	UF : 0, UT : 6,		CONFIG : 'N U T, 0, 0, 0',
	X =  94.552  mm,	Y =   -408.352  mm,	Z =   -258.182  mm,
	W =  90.000 deg,	P =   0.000 deg,	R =   90.000 deg
};
P[1225]{
   GP1:
	UF : 0, UT : 6,		CONFIG : 'N U T, 0, 0, 0',
	X =  95.294  mm,	Y =   -409.608  mm,	Z =   -258.283  mm,
	W =  90.000 deg,	P =   0.000 deg,	R =   90.000 deg
};
P[1226]{
   GP1:
	UF : 0, UT : 6,		CONFIG : 'N U T, 0, 0, 0',
	X =  95.758  mm,	Y =   -410.484  mm,	Z =   -258.027  mm,
	W =  90.000 deg,	P =   0.000 deg,	R =   90.000 deg
};
P[1227]{
   GP1:
	UF : 0, UT : 6,		CONFIG : 'N U T, 0, 0, 0',
	X =  97.788  mm,	Y =   -414.039  mm,	Z =   -257.885  mm,
	W =  90.000 deg,	P =   0.000 deg,	R =   90.000 deg
};
P[1228]{
   GP1:
	UF : 0, UT : 6,		CONFIG : 'N U T, 0, 0, 0',
	X =  98.420  mm,	Y =   -415.000  mm,	Z =   -258.363  mm,
	W =  90.000 deg,	P =   0.000 deg,	R =   90.000 deg
};
P[1229]{
   GP1:
	UF : 0, UT : 6,		CONFIG : 'N U T, 0, 0, 0',
	X =  98.908  mm,	Y =   -415.884  mm,	Z =   -258.225  mm,
	W =  90.000 deg,	P =   0.000 deg,	R =   90.000 deg
};
P[1230]{
   GP1:
	UF : 0, UT : 6,		CONFIG : 'N U T, 0, 0, 0',
	X =  99.222  mm,	Y =   -416.492  mm,	Z =   -257.998  mm,
	W =  90.000 deg,	P =   0.000 deg,	R =   90.000 deg
};
P[1231]{
   GP1:
	UF : 0, UT : 6,		CONFIG : 'N U T, 0, 0, 0',
	X =  99.637  mm,	Y =   -417.217  mm,	Z =   -257.979  mm,
	W =  90.000 deg,	P =   0.000 deg,	R =   90.000 deg
};
P[1232]{
   GP1:
	UF : 0, UT : 6,		CONFIG : 'N U T, 0, 0, 0',
	X =  100.678  mm,	Y =   -419.015  mm,	Z =   -257.989  mm,
	W =  90.000 deg,	P =   0.000 deg,	R =   90.000 deg
};
P[1233]{
   GP1:
	UF : 0, UT : 6,		CONFIG : 'N U T, 0, 0, 0',
	X =  102.165  mm,	Y =   -421.501  mm,	Z =   -258.308  mm,
	W =  90.000 deg,	P =   0.000 deg,	R =   90.000 deg
};
P[1234]{
   GP1:
	UF : 0, UT : 6,		CONFIG : 'N U T, 0, 0, 0',
	X =  102.557  mm,	Y =   -422.208  mm,	Z =   -258.207  mm,
	W =  90.000 deg,	P =   0.000 deg,	R =   90.000 deg
};
P[1235]{
   GP1:
	UF : 0, UT : 6,		CONFIG : 'N U T, 0, 0, 0',
	X =  103.682  mm,	Y =   -424.148  mm,	Z =   -258.237  mm,
	W =  90.000 deg,	P =   0.000 deg,	R =   90.000 deg
};
P[1236]{
   GP1:
	UF : 0, UT : 6,		CONFIG : 'N U T, 0, 0, 0',
	X =  104.838  mm,	Y =   -426.195  mm,	Z =   -258.076  mm,
	W =  90.000 deg,	P =   0.000 deg,	R =   90.000 deg
};
P[1237]{
   GP1:
	UF : 0, UT : 6,		CONFIG : 'N U T, 0, 0, 0',
	X =  106.776  mm,	Y =   -429.472  mm,	Z =   -258.366  mm,
	W =  90.000 deg,	P =   0.000 deg,	R =   90.000 deg
};
P[1238]{
   GP1:
	UF : 0, UT : 6,		CONFIG : 'N U T, 0, 0, 0',
	X =  107.228  mm,	Y =   -430.273  mm,	Z =   -258.299  mm,
	W =  90.000 deg,	P =   0.000 deg,	R =   90.000 deg
};
P[1239]{
   GP1:
	UF : 0, UT : 6,		CONFIG : 'N U T, 0, 0, 0',
	X =  108.043  mm,	Y =   -431.682  mm,	Z =   -258.309  mm,
	W =  90.000 deg,	P =   0.000 deg,	R =   90.000 deg
};
P[1240]{
   GP1:
	UF : 0, UT : 6,		CONFIG : 'N U T, 0, 0, 0',
	X =  108.614  mm,	Y =   -432.663  mm,	Z =   -258.336  mm,
	W =  90.000 deg,	P =   0.000 deg,	R =   90.000 deg
};
P[1241]{
   GP1:
	UF : 0, UT : 6,		CONFIG : 'N U T, 0, 0, 0',
	X =  110.290  mm,	Y =   -435.622  mm,	Z =   -258.135  mm,
	W =  90.000 deg,	P =   0.000 deg,	R =   90.000 deg
};
P[1242]{
   GP1:
	UF : 0, UT : 6,		CONFIG : 'N U T, 0, 0, 0',
	X =  110.941  mm,	Y =   -436.722  mm,	Z =   -258.230  mm,
	W =  90.000 deg,	P =   0.000 deg,	R =   90.000 deg
};
P[1243]{
   GP1:
	UF : 0, UT : 6,		CONFIG : 'N U T, 0, 0, 0',
	X =  112.232  mm,	Y =   -438.986  mm,	Z =   -258.130  mm,
	W =  90.000 deg,	P =   0.000 deg,	R =   90.000 deg
};
P[1244]{
   GP1:
	UF : 0, UT : 6,		CONFIG : 'N U T, 0, 0, 0',
	X =  113.189  mm,	Y =   -440.584  mm,	Z =   -258.341  mm,
	W =  90.000 deg,	P =   0.000 deg,	R =   90.000 deg
};
P[1245]{
   GP1:
	UF : 0, UT : 6,		CONFIG : 'N U T, 0, 0, 0',
	X =  114.856  mm,	Y =   -443.594  mm,	Z =   -257.910  mm,
	W =  90.000 deg,	P =   0.000 deg,	R =   90.000 deg
};
P[1246]{
   GP1:
	UF : 0, UT : 6,		CONFIG : 'N U T, 0, 0, 0',
	X =  115.439  mm,	Y =   -444.516  mm,	Z =   -258.220  mm,
	W =  90.000 deg,	P =   0.000 deg,	R =   90.000 deg
};
P[1247]{
   GP1:
	UF : 0, UT : 6,		CONFIG : 'N U T, 0, 0, 0',
	X =  115.884  mm,	Y =   -445.335  mm,	Z =   -258.046  mm,
	W =  90.000 deg,	P =   0.000 deg,	R =   90.000 deg
};
P[1248]{
   GP1:
	UF : 0, UT : 6,		CONFIG : 'N U T, 0, 0, 0',
	X =  116.583  mm,	Y =   -446.538  mm,	Z =   -258.073  mm,
	W =  90.000 deg,	P =   0.000 deg,	R =   90.000 deg
};
P[1249]{
   GP1:
	UF : 0, UT : 6,		CONFIG : 'N U T, 0, 0, 0',
	X =  117.265  mm,	Y =   -447.654  mm,	Z =   -258.308  mm,
	W =  90.000 deg,	P =   0.000 deg,	R =   90.000 deg
};
P[1250]{
   GP1:
	UF : 0, UT : 6,		CONFIG : 'N U T, 0, 0, 0',
	X =  118.172  mm,	Y =   -449.252  mm,	Z =   -258.213  mm,
	W =  90.000 deg,	P =   0.000 deg,	R =   90.000 deg
};
P[1251]{
   GP1:
	UF : 0, UT : 6,		CONFIG : 'N U T, 0, 0, 0',
	X =  119.589  mm,	Y =   -451.752  mm,	Z =   -258.047  mm,
	W =  90.000 deg,	P =   0.000 deg,	R =   90.000 deg
};
P[1252]{
   GP1:
	UF : 0, UT : 6,		CONFIG : 'N U T, 0, 0, 0',
	X =  120.416  mm,	Y =   -453.157  mm,	Z =   -258.146  mm,
	W =  90.000 deg,	P =   0.000 deg,	R =   90.000 deg
};
P[1253]{
   GP1:
	UF : 0, UT : 6,		CONFIG : 'N U T, 0, 0, 0',
	X =  120.901  mm,	Y =   -453.949  mm,	Z =   -258.320  mm,
	W =  90.000 deg,	P =   0.000 deg,	R =   90.000 deg
};
P[1254]{
   GP1:
	UF : 0, UT : 6,		CONFIG : 'N U T, 0, 0, 0',
	X =  121.824  mm,	Y =   -455.560  mm,	Z =   -258.271  mm,
	W =  90.000 deg,	P =   0.000 deg,	R =   90.000 deg
};
P[1255]{
   GP1:
	UF : 0, UT : 6,		CONFIG : 'N U T, 0, 0, 0',
	X =  122.704  mm,	Y =   -457.147  mm,	Z =   -258.049  mm,
	W =  90.000 deg,	P =   0.000 deg,	R =   90.000 deg
};
P[1256]{
   GP1:
	UF : 0, UT : 6,		CONFIG : 'N U T, 0, 0, 0',
	X =  123.451  mm,	Y =   -458.351  mm,	Z =   -258.366  mm,
	W =  90.000 deg,	P =   0.000 deg,	R =   90.000 deg
};
P[1257]{
   GP1:
	UF : 0, UT : 6,		CONFIG : 'N U T, 0, 0, 0',
	X =  124.051  mm,	Y =   -459.397  mm,	Z =   -258.345  mm,
	W =  90.000 deg,	P =   0.000 deg,	R =   90.000 deg
};
P[1258]{
   GP1:
	UF : 0, UT : 6,		CONFIG : 'N U T, 0, 0, 0',
	X =  125.157  mm,	Y =   -461.402  mm,	Z =   -258.020  mm,
	W =  90.000 deg,	P =   0.000 deg,	R =   90.000 deg
};
P[1259]{
   GP1:
	UF : 0, UT : 6,		CONFIG : 'N U T, 0, 0, 0',
	X =  127.066  mm,	Y =   -464.670  mm,	Z =   -258.163  mm,
	W =  90.000 deg,	P =   0.000 deg,	R =   90.000 deg
};
P[1260]{
   GP1:
	UF : 0, UT : 6,		CONFIG : 'N U T, 0, 0, 0',
	X =  128.906  mm,	Y =   -467.832  mm,	Z =   -258.243  mm,
	W =  90.000 deg,	P =   0.000 deg,	R =   90.000 deg
};
P[1261]{
   GP1:
	UF : 0, UT : 6,		CONFIG : 'N U T, 0, 0, 0',
	X =  130.187  mm,	Y =   -470.130  mm,	Z =   -257.965  mm,
	W =  90.000 deg,	P =   0.000 deg,	R =   90.000 deg
};
P[1262]{
   GP1:
	UF : 0, UT : 6,		CONFIG : 'N U T, 0, 0, 0',
	X =  133.362  mm,	Y =   -475.538  mm,	Z =   -258.285  mm,
	W =  90.000 deg,	P =   0.000 deg,	R =   90.000 deg
};
P[1263]{
   GP1:
	UF : 0, UT : 6,		CONFIG : 'N U T, 0, 0, 0',
	X =  134.419  mm,	Y =   -477.361  mm,	Z =   -258.319  mm,
	W =  90.000 deg,	P =   0.000 deg,	R =   90.000 deg
};
P[1264]{
   GP1:
	UF : 0, UT : 6,		CONFIG : 'N U T, 0, 0, 0',
	X =  135.215  mm,	Y =   -478.733  mm,	Z =   -258.340  mm,
	W =  90.000 deg,	P =   0.000 deg,	R =   90.000 deg
};
P[1265]{
   GP1:
	UF : 0, UT : 6,		CONFIG : 'N U T, 0, 0, 0',
	X =  135.836  mm,	Y =   -479.841  mm,	Z =   -258.224  mm,
	W =  90.000 deg,	P =   0.000 deg,	R =   90.000 deg
};
P[1266]{
   GP1:
	UF : 0, UT : 6,		CONFIG : 'N U T, 0, 0, 0',
	X =  136.333  mm,	Y =   -480.673  mm,	Z =   -258.327  mm,
	W =  90.000 deg,	P =   0.000 deg,	R =   90.000 deg
};
P[1267]{
   GP1:
	UF : 0, UT : 6,		CONFIG : 'N U T, 0, 0, 0',
	X =  136.704  mm,	Y =   -481.354  mm,	Z =   -258.194  mm,
	W =  90.000 deg,	P =   0.000 deg,	R =   90.000 deg
};
P[1268]{
   GP1:
	UF : 0, UT : 6,		CONFIG : 'N U T, 0, 0, 0',
	X =  137.629  mm,	Y =   -482.958  mm,	Z =   -258.179  mm,
	W =  90.000 deg,	P =   0.000 deg,	R =   90.000 deg
};
P[1269]{
   GP1:
	UF : 0, UT : 6,		CONFIG : 'N U T, 0, 0, 0',
	X =  137.961  mm,	Y =   -483.617  mm,	Z =   -257.886  mm,
	W =  90.000 deg,	P =   0.000 deg,	R =   90.000 deg
};
P[1270]{
   GP1:
	UF : 0, UT : 6,		CONFIG : 'N U T, 0, 0, 0',
	X =  138.519  mm,	Y =   -484.502  mm,	Z =   -258.173  mm,
	W =  90.000 deg,	P =   0.000 deg,	R =   90.000 deg
};
P[1271]{
   GP1:
	UF : 0, UT : 6,		CONFIG : 'N U T, 0, 0, 0',
	X =  139.565  mm,	Y =   -486.369  mm,	Z =   -257.974  mm,
	W =  90.000 deg,	P =   0.000 deg,	R =   90.000 deg
};
P[1272]{
   GP1:
	UF : 0, UT : 6,		CONFIG : 'N U T, 0, 0, 0',
	X =  140.108  mm,	Y =   -487.270  mm,	Z =   -258.117  mm,
	W =  90.000 deg,	P =   0.000 deg,	R =   90.000 deg
};
P[1273]{
   GP1:
	UF : 0, UT : 6,		CONFIG : 'N U T, 0, 0, 0',
	X =  140.575  mm,	Y =   -488.046  mm,	Z =   -258.234  mm,
	W =  90.000 deg,	P =   0.000 deg,	R =   90.000 deg
};
P[1274]{
   GP1:
	UF : 0, UT : 6,		CONFIG : 'N U T, 0, 0, 0',
	X =  140.969  mm,	Y =   -488.696  mm,	Z =   -258.351  mm,
	W =  90.000 deg,	P =   0.000 deg,	R =   90.000 deg
};
P[1275]{
   GP1:
	UF : 0, UT : 6,		CONFIG : 'N U T, 0, 0, 0',
	X =  142.429  mm,	Y =   -491.284  mm,	Z =   -258.141  mm,
	W =  90.000 deg,	P =   0.000 deg,	R =   90.000 deg
};
P[1276]{
   GP1:
	UF : 0, UT : 6,		CONFIG : 'N U T, 0, 0, 0',
	X =  143.194  mm,	Y =   -492.591  mm,	Z =   -258.201  mm,
	W =  90.000 deg,	P =   0.000 deg,	R =   90.000 deg
};
P[1277]{
   GP1:
	UF : 0, UT : 6,		CONFIG : 'N U T, 0, 0, 0',
	X =  143.776  mm,	Y =   -493.659  mm,	Z =   -257.984  mm,
	W =  90.000 deg,	P =   0.000 deg,	R =   90.000 deg
};
P[1278]{
   GP1:
	UF : 0, UT : 6,		CONFIG : 'N U T, 0, 0, 0',
	X =  146.005  mm,	Y =   -497.456  mm,	Z =   -258.215  mm,
	W =  90.000 deg,	P =   0.000 deg,	R =   90.000 deg
};
P[1279]{
   GP1:
	UF : 0, UT : 6,		CONFIG : 'N U T, 0, 0, 0',
	X =  146.357  mm,	Y =   -498.134  mm,	Z =   -257.971  mm,
	W =  90.000 deg,	P =   0.000 deg,	R =   90.000 deg
};
P[1280]{
   GP1:
	UF : 0, UT : 6,		CONFIG : 'N U T, 0, 0, 0',
	X =  146.841  mm,	Y =   -498.868  mm,	Z =   -258.337  mm,
	W =  90.000 deg,	P =   0.000 deg,	R =   90.000 deg
};
P[1281]{
   GP1:
	UF : 0, UT : 6,		CONFIG : 'N U T, 0, 0, 0',
	X =  148.554  mm,	Y =   -501.849  mm,	Z =   -258.294  mm,
	W =  90.000 deg,	P =   0.000 deg,	R =   90.000 deg
};
P[1282]{
   GP1:
	UF : 0, UT : 6,		CONFIG : 'N U T, 0, 0, 0',
	X =  149.699  mm,	Y =   -503.836  mm,	Z =   -258.269  mm,
	W =  90.000 deg,	P =   0.000 deg,	R =   90.000 deg
};
P[1283]{
   GP1:
	UF : 0, UT : 6,		CONFIG : 'N U T, 0, 0, 0',
	X =  150.552  mm,	Y =   -505.372  mm,	Z =   -258.067  mm,
	W =  90.000 deg,	P =   0.000 deg,	R =   90.000 deg
};
P[1284]{
   GP1:
	UF : 0, UT : 6,		CONFIG : 'N U T, 0, 0, 0',
	X =  151.351  mm,	Y =   -506.757  mm,	Z =   -258.063  mm,
	W =  90.000 deg,	P =   0.000 deg,	R =   90.000 deg
};
P[1285]{
   GP1:
	UF : 0, UT : 6,		CONFIG : 'N U T, 0, 0, 0',
	X =  153.612  mm,	Y =   -510.597  mm,	Z =   -258.330  mm,
	W =  90.000 deg,	P =   0.000 deg,	R =   90.000 deg
};
P[1286]{
   GP1:
	UF : 0, UT : 6,		CONFIG : 'N U T, 0, 0, 0',
	X =  155.200  mm,	Y =   -513.345  mm,	Z =   -258.341  mm,
	W =  90.000 deg,	P =   0.000 deg,	R =   90.000 deg
};
P[1287]{
   GP1:
	UF : 0, UT : 6,		CONFIG : 'N U T, 0, 0, 0',
	X =  156.191  mm,	Y =   -515.127  mm,	Z =   -258.111  mm,
	W =  90.000 deg,	P =   0.000 deg,	R =   90.000 deg
};
P[1288]{
   GP1:
	UF : 0, UT : 6,		CONFIG : 'N U T, 0, 0, 0',
	X =  156.669  mm,	Y =   -515.891  mm,	Z =   -258.331  mm,
	W =  90.000 deg,	P =   0.000 deg,	R =   90.000 deg
};
P[1289]{
   GP1:
	UF : 0, UT : 6,		CONFIG : 'N U T, 0, 0, 0',
	X =  157.149  mm,	Y =   -516.845  mm,	Z =   -257.901  mm,
	W =  90.000 deg,	P =   0.000 deg,	R =   90.000 deg
};
P[1290]{
   GP1:
	UF : 0, UT : 6,		CONFIG : 'N U T, 0, 0, 0',
	X =  157.848  mm,	Y =   -518.047  mm,	Z =   -257.931  mm,
	W =  90.000 deg,	P =   0.000 deg,	R =   90.000 deg
};
P[1291]{
   GP1:
	UF : 0, UT : 6,		CONFIG : 'N U T, 0, 0, 0',
	X =  158.394  mm,	Y =   -518.927  mm,	Z =   -258.161  mm,
	W =  90.000 deg,	P =   0.000 deg,	R =   90.000 deg
};
P[1292]{
   GP1:
	UF : 0, UT : 6,		CONFIG : 'N U T, 0, 0, 0',
	X =  159.080  mm,	Y =   -520.100  mm,	Z =   -258.219  mm,
	W =  90.000 deg,	P =   0.000 deg,	R =   90.000 deg
};
P[1293]{
   GP1:
	UF : 0, UT : 6,		CONFIG : 'N U T, 0, 0, 0',
	X =  159.685  mm,	Y =   -521.137  mm,	Z =   -258.258  mm,
	W =  90.000 deg,	P =   0.000 deg,	R =   90.000 deg
};
P[1294]{
   GP1:
	UF : 0, UT : 6,		CONFIG : 'N U T, 0, 0, 0',
	X =  160.896  mm,	Y =   -523.212  mm,	Z =   -258.336  mm,
	W =  90.000 deg,	P =   0.000 deg,	R =   90.000 deg
};
P[1295]{
   GP1:
	UF : 0, UT : 6,		CONFIG : 'N U T, 0, 0, 0',
	X =  161.420  mm,	Y =   -524.107  mm,	Z =   -258.373  mm,
	W =  90.000 deg,	P =   0.000 deg,	R =   90.000 deg
};
P[1296]{
   GP1:
	UF : 0, UT : 6,		CONFIG : 'N U T, 0, 0, 0',
	X =  162.073  mm,	Y =   -525.281  mm,	Z =   -258.223  mm,
	W =  90.000 deg,	P =   0.000 deg,	R =   90.000 deg
};
P[1297]{
   GP1:
	UF : 0, UT : 6,		CONFIG : 'N U T, 0, 0, 0',
	X =  162.748  mm,	Y =   -526.409  mm,	Z =   -258.372  mm,
	W =  90.000 deg,	P =   0.000 deg,	R =   90.000 deg
};
P[1298]{
   GP1:
	UF : 0, UT : 6,		CONFIG : 'N U T, 0, 0, 0',
	X =  163.531  mm,	Y =   -527.788  mm,	Z =   -258.291  mm,
	W =  90.000 deg,	P =   0.000 deg,	R =   90.000 deg
};
P[1299]{
   GP1:
	UF : 0, UT : 6,		CONFIG : 'N U T, 0, 0, 0',
	X =  164.056  mm,	Y =   -528.774  mm,	Z =   -258.018  mm,
	W =  90.000 deg,	P =   0.000 deg,	R =   90.000 deg
};
P[1300]{
   GP1:
	UF : 0, UT : 6,		CONFIG : 'N U T, 0, 0, 0',
	X =  165.402  mm,	Y =   -531.059  mm,	Z =   -257.928  mm,
	W =  90.000 deg,	P =   0.000 deg,	R =   90.000 deg
};
P[1301]{
   GP1:
	UF : 0, UT : 6,		CONFIG : 'N U T, 0, 0, 0',
	X =  171.437  mm,	Y =   -532.018  mm,	Z =   -257.891  mm,
	W =  90.000 deg,	P =   0.000 deg,	R =   90.000 deg
};
P[1302]{
   GP1:
	UF : 0, UT : 6,		CONFIG : 'N U T, 0, 0, 0',
	X =  173.114  mm,	Y =   -531.024  mm,	Z =   -258.050  mm,
	W =  90.000 deg,	P =   0.000 deg,	R =   90.000 deg
};
P[1303]{
   GP1:
	UF : 0, UT : 6,		CONFIG : 'N U T, 0, 0, 0',
	X =  174.297  mm,	Y =   -530.321  mm,	Z =   -258.173  mm,
	W =  90.000 deg,	P =   0.000 deg,	R =   90.000 deg
};
P[1304]{
   GP1:
	UF : 0, UT : 6,		CONFIG : 'N U T, 0, 0, 0',
	X =  177.321  mm,	Y =   -528.545  mm,	Z =   -258.360  mm,
	W =  90.000 deg,	P =   0.000 deg,	R =   90.000 deg
};
P[1305]{
   GP1:
	UF : 0, UT : 6,		CONFIG : 'N U T, 0, 0, 0',
	X =  179.891  mm,	Y =   -527.073  mm,	Z =   -258.279  mm,
	W =  90.000 deg,	P =   0.000 deg,	R =   90.000 deg
};
P[1306]{
   GP1:
	UF : 0, UT : 6,		CONFIG : 'N U T, 0, 0, 0',
	X =  181.912  mm,	Y =   -525.941  mm,	Z =   -258.067  mm,
	W =  90.000 deg,	P =   0.000 deg,	R =   90.000 deg
};
P[1307]{
   GP1:
	UF : 0, UT : 6,		CONFIG : 'N U T, 0, 0, 0',
	X =  183.221  mm,	Y =   -525.165  mm,	Z =   -258.193  mm,
	W =  90.000 deg,	P =   0.000 deg,	R =   90.000 deg
};
P[1308]{
   GP1:
	UF : 0, UT : 6,		CONFIG : 'N U T, 0, 0, 0',
	X =  184.975  mm,	Y =   -524.167  mm,	Z =   -258.100  mm,
	W =  90.000 deg,	P =   0.000 deg,	R =   90.000 deg
};
P[1309]{
   GP1:
	UF : 0, UT : 6,		CONFIG : 'N U T, 0, 0, 0',
	X =  185.658  mm,	Y =   -523.772  mm,	Z =   -258.108  mm,
	W =  90.000 deg,	P =   0.000 deg,	R =   90.000 deg
};
P[1310]{
   GP1:
	UF : 0, UT : 6,		CONFIG : 'N U T, 0, 0, 0',
	X =  186.905  mm,	Y =   -523.058  mm,	Z =   -258.068  mm,
	W =  90.000 deg,	P =   0.000 deg,	R =   90.000 deg
};
P[1311]{
   GP1:
	UF : 0, UT : 6,		CONFIG : 'N U T, 0, 0, 0',
	X =  188.208  mm,	Y =   -522.274  mm,	Z =   -258.263  mm,
	W =  90.000 deg,	P =   0.000 deg,	R =   90.000 deg
};
P[1312]{
   GP1:
	UF : 0, UT : 6,		CONFIG : 'N U T, 0, 0, 0',
	X =  189.957  mm,	Y =   -521.293  mm,	Z =   -258.086  mm,
	W =  90.000 deg,	P =   0.000 deg,	R =   90.000 deg
};
P[1313]{
   GP1:
	UF : 0, UT : 6,		CONFIG : 'N U T, 0, 0, 0',
	X =  190.680  mm,	Y =   -520.845  mm,	Z =   -258.275  mm,
	W =  90.000 deg,	P =   0.000 deg,	R =   90.000 deg
};
P[1314]{
   GP1:
	UF : 0, UT : 6,		CONFIG : 'N U T, 0, 0, 0',
	X =  194.586  mm,	Y =   -518.623  mm,	Z =   -258.070  mm,
	W =  90.000 deg,	P =   0.000 deg,	R =   90.000 deg
};
P[1315]{
   GP1:
	UF : 0, UT : 6,		CONFIG : 'N U T, 0, 0, 0',
	X =  195.213  mm,	Y =   -518.258  mm,	Z =   -258.088  mm,
	W =  90.000 deg,	P =   0.000 deg,	R =   90.000 deg
};
P[1316]{
   GP1:
	UF : 0, UT : 6,		CONFIG : 'N U T, 0, 0, 0',
	X =  196.243  mm,	Y =   -517.658  mm,	Z =   -258.119  mm,
	W =  90.000 deg,	P =   0.000 deg,	R =   90.000 deg
};
P[1317]{
   GP1:
	UF : 0, UT : 6,		CONFIG : 'N U T, 0, 0, 0',
	X =  197.152  mm,	Y =   -517.171  mm,	Z =   -257.888  mm,
	W =  90.000 deg,	P =   0.000 deg,	R =   90.000 deg
};
P[1318]{
   GP1:
	UF : 0, UT : 6,		CONFIG : 'N U T, 0, 0, 0',
	X =  198.227  mm,	Y =   -516.501  mm,	Z =   -258.195  mm,
	W =  90.000 deg,	P =   0.000 deg,	R =   90.000 deg
};
P[1319]{
   GP1:
	UF : 0, UT : 6,		CONFIG : 'N U T, 0, 0, 0',
	X =  198.898  mm,	Y =   -516.139  mm,	Z =   -258.033  mm,
	W =  90.000 deg,	P =   0.000 deg,	R =   90.000 deg
};
P[1320]{
   GP1:
	UF : 0, UT : 6,		CONFIG : 'N U T, 0, 0, 0',
	X =  200.146  mm,	Y =   -515.419  mm,	Z =   -258.027  mm,
	W =  90.000 deg,	P =   0.000 deg,	R =   90.000 deg
};
P[1321]{
   GP1:
	UF : 0, UT : 6,		CONFIG : 'N U T, 0, 0, 0',
	X =  200.957  mm,	Y =   -514.922  mm,	Z =   -258.211  mm,
	W =  90.000 deg,	P =   0.000 deg,	R =   90.000 deg
};
P[1322]{
   GP1:
	UF : 0, UT : 6,		CONFIG : 'N U T, 0, 0, 0',
	X =  202.094  mm,	Y =   -514.264  mm,	Z =   -258.222  mm,
	W =  90.000 deg,	P =   0.000 deg,	R =   90.000 deg
};
P[1323]{
   GP1:
	UF : 0, UT : 6,		CONFIG : 'N U T, 0, 0, 0',
	X =  203.821  mm,	Y =   -513.312  mm,	Z =   -257.937  mm,
	W =  90.000 deg,	P =   0.000 deg,	R =   90.000 deg
};
P[1324]{
   GP1:
	UF : 0, UT : 6,		CONFIG : 'N U T, 0, 0, 0',
	X =  204.474  mm,	Y =   -512.873  mm,	Z =   -258.316  mm,
	W =  90.000 deg,	P =   0.000 deg,	R =   90.000 deg
};
P[1325]{
   GP1:
	UF : 0, UT : 6,		CONFIG : 'N U T, 0, 0, 0',
	X =  207.804  mm,	Y =   -510.983  mm,	Z =   -258.119  mm,
	W =  90.000 deg,	P =   0.000 deg,	R =   90.000 deg
};
P[1326]{
   GP1:
	UF : 0, UT : 6,		CONFIG : 'N U T, 0, 0, 0',
	X =  211.478  mm,	Y =   -508.873  mm,	Z =   -258.051  mm,
	W =  90.000 deg,	P =   0.000 deg,	R =   90.000 deg
};
P[1327]{
   GP1:
	UF : 0, UT : 6,		CONFIG : 'N U T, 0, 0, 0',
	X =  213.146  mm,	Y =   -507.925  mm,	Z =   -257.957  mm,
	W =  90.000 deg,	P =   0.000 deg,	R =   90.000 deg
};
P[1328]{
   GP1:
	UF : 0, UT : 6,		CONFIG : 'N U T, 0, 0, 0',
	X =  215.809  mm,	Y =   -506.372  mm,	Z =   -258.046  mm,
	W =  90.000 deg,	P =   0.000 deg,	R =   90.000 deg
};
P[1329]{
   GP1:
	UF : 0, UT : 6,		CONFIG : 'N U T, 0, 0, 0',
	X =  216.662  mm,	Y =   -505.833  mm,	Z =   -258.335  mm,
	W =  90.000 deg,	P =   0.000 deg,	R =   90.000 deg
};
P[1330]{
   GP1:
	UF : 0, UT : 6,		CONFIG : 'N U T, 0, 0, 0',
	X =  217.248  mm,	Y =   -505.564  mm,	Z =   -257.912  mm,
	W =  90.000 deg,	P =   0.000 deg,	R =   90.000 deg
};
P[1331]{
   GP1:
	UF : 0, UT : 6,		CONFIG : 'N U T, 0, 0, 0',
	X =  218.979  mm,	Y =   -504.496  mm,	Z =   -258.335  mm,
	W =  90.000 deg,	P =   0.000 deg,	R =   90.000 deg
};
P[1332]{
   GP1:
	UF : 0, UT : 6,		CONFIG : 'N U T, 0, 0, 0',
	X =  219.768  mm,	Y =   -504.089  mm,	Z =   -258.034  mm,
	W =  90.000 deg,	P =   0.000 deg,	R =   90.000 deg
};
P[1333]{
   GP1:
	UF : 0, UT : 6,		CONFIG : 'N U T, 0, 0, 0',
	X =  221.190  mm,	Y =   -503.284  mm,	Z =   -257.934  mm,
	W =  90.000 deg,	P =   0.000 deg,	R =   90.000 deg
};
P[1334]{
   GP1:
	UF : 0, UT : 6,		CONFIG : 'N U T, 0, 0, 0',
	X =  222.943  mm,	Y =   -502.222  mm,	Z =   -258.247  mm,
	W =  90.000 deg,	P =   0.000 deg,	R =   90.000 deg
};
P[1335]{
   GP1:
	UF : 0, UT : 6,		CONFIG : 'N U T, 0, 0, 0',
	X =  225.305  mm,	Y =   -500.841  mm,	Z =   -258.341  mm,
	W =  90.000 deg,	P =   0.000 deg,	R =   90.000 deg
};
P[1336]{
   GP1:
	UF : 0, UT : 6,		CONFIG : 'N U T, 0, 0, 0',
	X =  228.005  mm,	Y =   -499.324  mm,	Z =   -258.090  mm,
	W =  90.000 deg,	P =   0.000 deg,	R =   90.000 deg
};
P[1337]{
   GP1:
	UF : 0, UT : 6,		CONFIG : 'N U T, 0, 0, 0',
	X =  230.940  mm,	Y =   -497.594  mm,	Z =   -258.312  mm,
	W =  90.000 deg,	P =   0.000 deg,	R =   90.000 deg
};
P[1338]{
   GP1:
	UF : 0, UT : 6,		CONFIG : 'N U T, 0, 0, 0',
	X =  233.189  mm,	Y =   -496.307  mm,	Z =   -258.239  mm,
	W =  90.000 deg,	P =   0.000 deg,	R =   90.000 deg
};
P[1339]{
   GP1:
	UF : 0, UT : 6,		CONFIG : 'N U T, 0, 0, 0',
	X =  234.235  mm,	Y =   -495.696  mm,	Z =   -258.275  mm,
	W =  90.000 deg,	P =   0.000 deg,	R =   90.000 deg
};
P[1340]{
   GP1:
	UF : 0, UT : 6,		CONFIG : 'N U T, 0, 0, 0',
	X =  235.419  mm,	Y =   -495.018  mm,	Z =   -258.243  mm,
	W =  90.000 deg,	P =   0.000 deg,	R =   90.000 deg
};
P[1341]{
   GP1:
	UF : 0, UT : 6,		CONFIG : 'N U T, 0, 0, 0',
	X =  238.703  mm,	Y =   -493.142  mm,	Z =   -258.118  mm,
	W =  90.000 deg,	P =   0.000 deg,	R =   90.000 deg
};
P[1342]{
   GP1:
	UF : 0, UT : 6,		CONFIG : 'N U T, 0, 0, 0',
	X =  239.544  mm,	Y =   -492.670  mm,	Z =   -258.032  mm,
	W =  90.000 deg,	P =   0.000 deg,	R =   90.000 deg
};
P[1343]{
   GP1:
	UF : 0, UT : 6,		CONFIG : 'N U T, 0, 0, 0',
	X =  241.793  mm,	Y =   -491.361  mm,	Z =   -258.099  mm,
	W =  90.000 deg,	P =   0.000 deg,	R =   90.000 deg
};
P[1344]{
   GP1:
	UF : 0, UT : 6,		CONFIG : 'N U T, 0, 0, 0',
	X =  243.548  mm,	Y =   -490.371  mm,	Z =   -257.961  mm,
	W =  90.000 deg,	P =   0.000 deg,	R =   90.000 deg
};
P[1345]{
   GP1:
	UF : 0, UT : 6,		CONFIG : 'N U T, 0, 0, 0',
	X =  244.521  mm,	Y =   -489.803  mm,	Z =   -257.994  mm,
	W =  90.000 deg,	P =   0.000 deg,	R =   90.000 deg
};
P[1346]{
   GP1:
	UF : 0, UT : 6,		CONFIG : 'N U T, 0, 0, 0',
	X =  246.068  mm,	Y =   -488.882  mm,	Z =   -258.168  mm,
	W =  90.000 deg,	P =   0.000 deg,	R =   90.000 deg
};
P[1347]{
   GP1:
	UF : 0, UT : 6,		CONFIG : 'N U T, 0, 0, 0',
	X =  247.393  mm,	Y =   -488.086  mm,	Z =   -258.360  mm,
	W =  90.000 deg,	P =   0.000 deg,	R =   90.000 deg
};
P[1348]{
   GP1:
	UF : 0, UT : 6,		CONFIG : 'N U T, 0, 0, 0',
	X =  251.159  mm,	Y =   -485.919  mm,	Z =   -258.311  mm,
	W =  90.000 deg,	P =   0.000 deg,	R =   90.000 deg
};
P[1349]{
   GP1:
	UF : 0, UT : 6,		CONFIG : 'N U T, 0, 0, 0',
	X =  252.384  mm,	Y =   -485.203  mm,	Z =   -258.369  mm,
	W =  90.000 deg,	P =   0.000 deg,	R =   90.000 deg
};
P[1350]{
   GP1:
	UF : 0, UT : 6,		CONFIG : 'N U T, 0, 0, 0',
	X =  253.645  mm,	Y =   -484.525  mm,	Z =   -258.052  mm,
	W =  90.000 deg,	P =   0.000 deg,	R =   90.000 deg
};
P[1351]{
   GP1:
	UF : 0, UT : 6,		CONFIG : 'N U T, 0, 0, 0',
	X =  254.710  mm,	Y =   -483.906  mm,	Z =   -258.082  mm,
	W =  90.000 deg,	P =   0.000 deg,	R =   90.000 deg
};
P[1352]{
   GP1:
	UF : 0, UT : 6,		CONFIG : 'N U T, 0, 0, 0',
	X =  256.308  mm,	Y =   -482.938  mm,	Z =   -258.359  mm,
	W =  90.000 deg,	P =   0.000 deg,	R =   90.000 deg
};
P[1353]{
   GP1:
	UF : 0, UT : 6,		CONFIG : 'N U T, 0, 0, 0',
	X =  257.640  mm,	Y =   -482.175  mm,	Z =   -258.324  mm,
	W =  90.000 deg,	P =   0.000 deg,	R =   90.000 deg
};
P[1354]{
   GP1:
	UF : 0, UT : 6,		CONFIG : 'N U T, 0, 0, 0',
	X =  259.031  mm,	Y =   -481.402  mm,	Z =   -258.140  mm,
	W =  90.000 deg,	P =   0.000 deg,	R =   90.000 deg
};
P[1355]{
   GP1:
	UF : 0, UT : 6,		CONFIG : 'N U T, 0, 0, 0',
	X =  260.378  mm,	Y =   -480.662  mm,	Z =   -257.903  mm,
	W =  90.000 deg,	P =   0.000 deg,	R =   90.000 deg
};
P[1356]{
   GP1:
	UF : 0, UT : 6,		CONFIG : 'N U T, 0, 0, 0',
	X =  261.945  mm,	Y =   -479.747  mm,	Z =   -257.970  mm,
	W =  90.000 deg,	P =   0.000 deg,	R =   90.000 deg
};
P[1357]{
   GP1:
	UF : 0, UT : 6,		CONFIG : 'N U T, 0, 0, 0',
	X =  263.572  mm,	Y =   -478.763  mm,	Z =   -258.245  mm,
	W =  90.000 deg,	P =   0.000 deg,	R =   90.000 deg
};
P[1358]{
   GP1:
	UF : 0, UT : 6,		CONFIG : 'N U T, 0, 0, 0',
	X =  265.019  mm,	Y =   -477.944  mm,	Z =   -258.140  mm,
	W =  90.000 deg,	P =   0.000 deg,	R =   90.000 deg
};
P[1359]{
   GP1:
	UF : 0, UT : 6,		CONFIG : 'N U T, 0, 0, 0',
	X =  265.912  mm,	Y =   -477.435  mm,	Z =   -258.099  mm,
	W =  90.000 deg,	P =   0.000 deg,	R =   90.000 deg
};
P[1360]{
   GP1:
	UF : 0, UT : 6,		CONFIG : 'N U T, 0, 0, 0',
	X =  268.353  mm,	Y =   -476.034  mm,	Z =   -258.047  mm,
	W =  90.000 deg,	P =   0.000 deg,	R =   90.000 deg
};
P[1361]{
   GP1:
	UF : 0, UT : 6,		CONFIG : 'N U T, 0, 0, 0',
	X =  268.952  mm,	Y =   -475.658  mm,	Z =   -258.240  mm,
	W =  90.000 deg,	P =   0.000 deg,	R =   90.000 deg
};
P[1362]{
   GP1:
	UF : 0, UT : 6,		CONFIG : 'N U T, 0, 0, 0',
	X =  269.997  mm,	Y =   -475.072  mm,	Z =   -258.130  mm,
	W =  90.000 deg,	P =   0.000 deg,	R =   90.000 deg
};
P[1363]{
   GP1:
	UF : 0, UT : 6,		CONFIG : 'N U T, 0, 0, 0',
	X =  270.885  mm,	Y =   -474.539  mm,	Z =   -258.252  mm,
	W =  90.000 deg,	P =   0.000 deg,	R =   90.000 deg
};
P[1364]{
   GP1:
	UF : 0, UT : 6,		CONFIG : 'N U T, 0, 0, 0',
	X =  271.725  mm,	Y =   -474.059  mm,	Z =   -258.217  mm,
	W =  90.000 deg,	P =   0.000 deg,	R =   90.000 deg
};
P[1365]{
   GP1:
	UF : 0, UT : 6,		CONFIG : 'N U T, 0, 0, 0',
	X =  272.377  mm,	Y =   -473.666  mm,	Z =   -258.326  mm,
	W =  90.000 deg,	P =   0.000 deg,	R =   90.000 deg
};
P[1366]{
   GP1:
	UF : 0, UT : 6,		CONFIG : 'N U T, 0, 0, 0',
	X =  273.202  mm,	Y =   -473.234  mm,	Z =   -258.051  mm,
	W =  90.000 deg,	P =   0.000 deg,	R =   90.000 deg
};
P[1367]{
   GP1:
	UF : 0, UT : 6,		CONFIG : 'N U T, 0, 0, 0',
	X =  274.534  mm,	Y =   -472.486  mm,	Z =   -257.914  mm,
	W =  90.000 deg,	P =   0.000 deg,	R =   90.000 deg
};
P[1368]{
   GP1:
	UF : 0, UT : 6,		CONFIG : 'N U T, 0, 0, 0',
	X =  275.485  mm,	Y =   -471.873  mm,	Z =   -258.319  mm,
	W =  90.000 deg,	P =   0.000 deg,	R =   90.000 deg
};
P[1369]{
   GP1:
	UF : 0, UT : 6,		CONFIG : 'N U T, 0, 0, 0',
	X =  278.237  mm,	Y =   -470.286  mm,	Z =   -258.303  mm,
	W =  90.000 deg,	P =   0.000 deg,	R =   90.000 deg
};
P[1370]{
   GP1:
	UF : 0, UT : 6,		CONFIG : 'N U T, 0, 0, 0',
	X =  279.547  mm,	Y =   -469.538  mm,	Z =   -258.251  mm,
	W =  90.000 deg,	P =   0.000 deg,	R =   90.000 deg
};
P[1371]{
   GP1:
	UF : 0, UT : 6,		CONFIG : 'N U T, 0, 0, 0',
	X =  280.823  mm,	Y =   -468.788  mm,	Z =   -258.334  mm,
	W =  90.000 deg,	P =   0.000 deg,	R =   90.000 deg
};
P[1372]{
   GP1:
	UF : 0, UT : 6,		CONFIG : 'N U T, 0, 0, 0',
	X =  281.865  mm,	Y =   -468.192  mm,	Z =   -258.297  mm,
	W =  90.000 deg,	P =   0.000 deg,	R =   90.000 deg
};
P[1373]{
   GP1:
	UF : 0, UT : 6,		CONFIG : 'N U T, 0, 0, 0',
	X =  283.101  mm,	Y =   -467.511  mm,	Z =   -258.097  mm,
	W =  90.000 deg,	P =   0.000 deg,	R =   90.000 deg
};
P[1374]{
   GP1:
	UF : 0, UT : 6,		CONFIG : 'N U T, 0, 0, 0',
	X =  283.694  mm,	Y =   -467.169  mm,	Z =   -258.093  mm,
	W =  90.000 deg,	P =   0.000 deg,	R =   90.000 deg
};
P[1375]{
   GP1:
	UF : 0, UT : 6,		CONFIG : 'N U T, 0, 0, 0',
	X =  284.792  mm,	Y =   -466.524  mm,	Z =   -258.162  mm,
	W =  90.000 deg,	P =   0.000 deg,	R =   90.000 deg
};
P[1376]{
   GP1:
	UF : 0, UT : 6,		CONFIG : 'N U T, 0, 0, 0',
	X =  286.844  mm,	Y =   -465.339  mm,	Z =   -258.165  mm,
	W =  90.000 deg,	P =   0.000 deg,	R =   90.000 deg
};
P[1377]{
   GP1:
	UF : 0, UT : 6,		CONFIG : 'N U T, 0, 0, 0',
	X =  287.815  mm,	Y =   -464.787  mm,	Z =   -258.105  mm,
	W =  90.000 deg,	P =   0.000 deg,	R =   90.000 deg
};
P[1378]{
   GP1:
	UF : 0, UT : 6,		CONFIG : 'N U T, 0, 0, 0',
	X =  288.412  mm,	Y =   -464.410  mm,	Z =   -258.305  mm,
	W =  90.000 deg,	P =   0.000 deg,	R =   90.000 deg
};
P[1379]{
   GP1:
	UF : 0, UT : 6,		CONFIG : 'N U T, 0, 0, 0',
	X =  290.305  mm,	Y =   -463.352  mm,	Z =   -258.096  mm,
	W =  90.000 deg,	P =   0.000 deg,	R =   90.000 deg
};
P[1380]{
   GP1:
	UF : 0, UT : 6,		CONFIG : 'N U T, 0, 0, 0',
	X =  290.933  mm,	Y =   -462.977  mm,	Z =   -258.169  mm,
	W =  90.000 deg,	P =   0.000 deg,	R =   90.000 deg
};
P[1381]{
   GP1:
	UF : 0, UT : 6,		CONFIG : 'N U T, 0, 0, 0',
	X =  291.705  mm,	Y =   -462.568  mm,	Z =   -257.946  mm,
	W =  90.000 deg,	P =   0.000 deg,	R =   90.000 deg
};
P[1382]{
   GP1:
	UF : 0, UT : 6,		CONFIG : 'N U T, 0, 0, 0',
	X =  293.001  mm,	Y =   -461.770  mm,	Z =   -258.253  mm,
	W =  90.000 deg,	P =   0.000 deg,	R =   90.000 deg
};
P[1383]{
   GP1:
	UF : 0, UT : 6,		CONFIG : 'N U T, 0, 0, 0',
	X =  293.996  mm,	Y =   -461.175  mm,	Z =   -258.376  mm,
	W =  90.000 deg,	P =   0.000 deg,	R =   90.000 deg
};
P[1384]{
   GP1:
	UF : 0, UT : 6,		CONFIG : 'N U T, 0, 0, 0',
	X =  296.393  mm,	Y =   -459.795  mm,	Z =   -258.350  mm,
	W =  90.000 deg,	P =   0.000 deg,	R =   90.000 deg
};
P[1385]{
   GP1:
	UF : 0, UT : 6,		CONFIG : 'N U T, 0, 0, 0',
	X =  297.026  mm,	Y =   -459.435  mm,	Z =   -258.320  mm,
	W =  90.000 deg,	P =   0.000 deg,	R =   90.000 deg
};
P[1386]{
   GP1:
	UF : 0, UT : 6,		CONFIG : 'N U T, 0, 0, 0',
	X =  298.733  mm,	Y =   -458.463  mm,	Z =   -258.230  mm,
	W =  90.000 deg,	P =   0.000 deg,	R =   90.000 deg
};
P[1387]{
   GP1:
	UF : 0, UT : 6,		CONFIG : 'N U T, 0, 0, 0',
	X =  299.648  mm,	Y =   -457.952  mm,	Z =   -258.125  mm,
	W =  90.000 deg,	P =   0.000 deg,	R =   90.000 deg
};
P[1388]{
   GP1:
	UF : 0, UT : 6,		CONFIG : 'N U T, 0, 0, 0',
	X =  300.684  mm,	Y =   -457.374  mm,	Z =   -258.005  mm,
	W =  90.000 deg,	P =   0.000 deg,	R =   90.000 deg
};
P[1389]{
   GP1:
	UF : 0, UT : 6,		CONFIG : 'N U T, 0, 0, 0',
	X =  301.364  mm,	Y =   -456.978  mm,	Z =   -258.024  mm,
	W =  90.000 deg,	P =   0.000 deg,	R =   90.000 deg
};
P[1390]{
   GP1:
	UF : 0, UT : 6,		CONFIG : 'N U T, 0, 0, 0',
	X =  302.193  mm,	Y =   -456.471  mm,	Z =   -258.203  mm,
	W =  90.000 deg,	P =   0.000 deg,	R =   90.000 deg
};
P[1391]{
   GP1:
	UF : 0, UT : 6,		CONFIG : 'N U T, 0, 0, 0',
	X =  302.812  mm,	Y =   -456.115  mm,	Z =   -258.185  mm,
	W =  90.000 deg,	P =   0.000 deg,	R =   90.000 deg
};
P[1392]{
   GP1:
	UF : 0, UT : 6,		CONFIG : 'N U T, 0, 0, 0',
	X =  303.595  mm,	Y =   -455.655  mm,	Z =   -258.241  mm,
	W =  90.000 deg,	P =   0.000 deg,	R =   90.000 deg
};
P[1393]{
   GP1:
	UF : 0, UT : 6,		CONFIG : 'N U T, 0, 0, 0',
	X =  304.735  mm,	Y =   -455.034  mm,	Z =   -258.008  mm,
	W =  90.000 deg,	P =   0.000 deg,	R =   90.000 deg
};
P[1394]{
   GP1:
	UF : 0, UT : 6,		CONFIG : 'N U T, 0, 0, 0',
	X =  305.734  mm,	Y =   -454.454  mm,	Z =   -258.027  mm,
	W =  90.000 deg,	P =   0.000 deg,	R =   90.000 deg
};
P[1395]{
   GP1:
	UF : 0, UT : 6,		CONFIG : 'N U T, 0, 0, 0',
	X =  307.496  mm,	Y =   -453.423  mm,	Z =   -258.114  mm,
	W =  90.000 deg,	P =   0.000 deg,	R =   90.000 deg
};
P[1396]{
   GP1:
	UF : 0, UT : 6,		CONFIG : 'N U T, 0, 0, 0',
	X =  310.657  mm,	Y =   -451.558  mm,	Z =   -258.358  mm,
	W =  90.000 deg,	P =   0.000 deg,	R =   90.000 deg
};
P[1397]{
   GP1:
	UF : 0, UT : 6,		CONFIG : 'N U T, 0, 0, 0',
	X =  311.623  mm,	Y =   -451.038  mm,	Z =   -258.126  mm,
	W =  90.000 deg,	P =   0.000 deg,	R =   90.000 deg
};
P[1398]{
   GP1:
	UF : 0, UT : 6,		CONFIG : 'N U T, 0, 0, 0',
	X =  312.842  mm,	Y =   -450.311  mm,	Z =   -258.270  mm,
	W =  90.000 deg,	P =   0.000 deg,	R =   90.000 deg
};
P[1399]{
   GP1:
	UF : 0, UT : 6,		CONFIG : 'N U T, 0, 0, 0',
	X =  314.065  mm,	Y =   -449.605  mm,	Z =   -258.270  mm,
	W =  90.000 deg,	P =   0.000 deg,	R =   90.000 deg
};
P[1400]{
   GP1:
	UF : 0, UT : 6,		CONFIG : 'N U T, 0, 0, 0',
	X =  315.646  mm,	Y =   -448.717  mm,	Z =   -258.111  mm,
	W =  90.000 deg,	P =   0.000 deg,	R =   90.000 deg
};
P[1401]{
   GP1:
	UF : 0, UT : 6,		CONFIG : 'N U T, 0, 0, 0',
	X =  317.171  mm,	Y =   -447.825  mm,	Z =   -258.180  mm,
	W =  90.000 deg,	P =   0.000 deg,	R =   90.000 deg
};
P[1402]{
   GP1:
	UF : 0, UT : 6,		CONFIG : 'N U T, 0, 0, 0',
	X =  321.164  mm,	Y =   -445.517  mm,	Z =   -258.199  mm,
	W =  90.000 deg,	P =   0.000 deg,	R =   90.000 deg
};
P[1403]{
   GP1:
	UF : 0, UT : 6,		CONFIG : 'N U T, 0, 0, 0',
	X =  324.345  mm,	Y =   -443.699  mm,	Z =   -258.082  mm,
	W =  90.000 deg,	P =   0.000 deg,	R =   90.000 deg
};
P[1404]{
   GP1:
	UF : 0, UT : 6,		CONFIG : 'N U T, 0, 0, 0',
	X =  326.731  mm,	Y =   -442.289  mm,	Z =   -258.282  mm,
	W =  90.000 deg,	P =   0.000 deg,	R =   90.000 deg
};
P[1405]{
   GP1:
	UF : 0, UT : 6,		CONFIG : 'N U T, 0, 0, 0',
	X =  329.901  mm,	Y =   -440.494  mm,	Z =   -258.065  mm,
	W =  90.000 deg,	P =   0.000 deg,	R =   90.000 deg
};
P[1406]{
   GP1:
	UF : 0, UT : 6,		CONFIG : 'N U T, 0, 0, 0',
	X =  330.790  mm,	Y =   -439.989  mm,	Z =   -258.018  mm,
	W =  90.000 deg,	P =   0.000 deg,	R =   90.000 deg
};
P[1407]{
   GP1:
	UF : 0, UT : 6,		CONFIG : 'N U T, 0, 0, 0',
	X =  331.434  mm,	Y =   -439.565  mm,	Z =   -258.340  mm,
	W =  90.000 deg,	P =   0.000 deg,	R =   90.000 deg
};
P[1408]{
   GP1:
	UF : 0, UT : 6,		CONFIG : 'N U T, 0, 0, 0',
	X =  332.220  mm,	Y =   -439.153  mm,	Z =   -258.082  mm,
	W =  90.000 deg,	P =   0.000 deg,	R =   90.000 deg
};
P[1409]{
   GP1:
	UF : 0, UT : 6,		CONFIG : 'N U T, 0, 0, 0',
	X =  333.473  mm,	Y =   -438.445  mm,	Z =   -257.980  mm,
	W =  90.000 deg,	P =   0.000 deg,	R =   90.000 deg
};
P[1410]{
   GP1:
	UF : 0, UT : 6,		CONFIG : 'N U T, 0, 0, 0',
	X =  334.443  mm,	Y =   -437.850  mm,	Z =   -258.199  mm,
	W =  90.000 deg,	P =   0.000 deg,	R =   90.000 deg
};
P[1411]{
   GP1:
	UF : 0, UT : 6,		CONFIG : 'N U T, 0, 0, 0',
	X =  336.657  mm,	Y =   -436.551  mm,	Z =   -258.322  mm,
	W =  90.000 deg,	P =   0.000 deg,	R =   90.000 deg
};
P[1412]{
   GP1:
	UF : 0, UT : 6,		CONFIG : 'N U T, 0, 0, 0',
	X =  338.195  mm,	Y =   -435.703  mm,	Z =   -258.082  mm,
	W =  90.000 deg,	P =   0.000 deg,	R =   90.000 deg
};
P[1413]{
   GP1:
	UF : 0, UT : 6,		CONFIG : 'N U T, 0, 0, 0',
	X =  341.077  mm,	Y =   -433.998  mm,	Z =   -258.330  mm,
	W =  90.000 deg,	P =   0.000 deg,	R =   90.000 deg
};
P[1414]{
   GP1:
	UF : 0, UT : 6,		CONFIG : 'N U T, 0, 0, 0',
	X =  343.418  mm,	Y =   -432.658  mm,	Z =   -258.258  mm,
	W =  90.000 deg,	P =   0.000 deg,	R =   90.000 deg
};
P[1415]{
   GP1:
	UF : 0, UT : 6,		CONFIG : 'N U T, 0, 0, 0',
	X =  345.775  mm,	Y =   -431.295  mm,	Z =   -258.273  mm,
	W =  90.000 deg,	P =   0.000 deg,	R =   90.000 deg
};
P[1416]{
   GP1:
	UF : 0, UT : 6,		CONFIG : 'N U T, 0, 0, 0',
	X =  346.718  mm,	Y =   -430.737  mm,	Z =   -258.358  mm,
	W =  90.000 deg,	P =   0.000 deg,	R =   90.000 deg
};
P[1417]{
   GP1:
	UF : 0, UT : 6,		CONFIG : 'N U T, 0, 0, 0',
	X =  347.784  mm,	Y =   -430.186  mm,	Z =   -257.954  mm,
	W =  90.000 deg,	P =   0.000 deg,	R =   90.000 deg
};
P[1418]{
   GP1:
	UF : 0, UT : 6,		CONFIG : 'N U T, 0, 0, 0',
	X =  350.692  mm,	Y =   -428.471  mm,	Z =   -258.177  mm,
	W =  90.000 deg,	P =   0.000 deg,	R =   90.000 deg
};
P[1419]{
   GP1:
	UF : 0, UT : 6,		CONFIG : 'N U T, 0, 0, 0',
	X =  352.922  mm,	Y =   -427.165  mm,	Z =   -258.293  mm,
	W =  90.000 deg,	P =   0.000 deg,	R =   90.000 deg
};
P[1420]{
   GP1:
	UF : 0, UT : 6,		CONFIG : 'N U T, 0, 0, 0',
	X =  353.853  mm,	Y =   -426.616  mm,	Z =   -258.360  mm,
	W =  90.000 deg,	P =   0.000 deg,	R =   90.000 deg
};
P[1421]{
   GP1:
	UF : 0, UT : 6,		CONFIG : 'N U T, 0, 0, 0',
	X =  354.660  mm,	Y =   -426.153  mm,	Z =   -258.344  mm,
	W =  90.000 deg,	P =   0.000 deg,	R =   90.000 deg
};
P[1422]{
   GP1:
	UF : 0, UT : 6,		CONFIG : 'N U T, 0, 0, 0',
	X =  357.272  mm,	Y =   -424.677  mm,	Z =   -258.148  mm,
	W =  90.000 deg,	P =   0.000 deg,	R =   90.000 deg
};
P[1423]{
   GP1:
	UF : 0, UT : 6,		CONFIG : 'N U T, 0, 0, 0',
	X =  359.723  mm,	Y =   -423.259  mm,	Z =   -258.169  mm,
	W =  90.000 deg,	P =   0.000 deg,	R =   90.000 deg
};
P[1424]{
   GP1:
	UF : 0, UT : 6,		CONFIG : 'N U T, 0, 0, 0',
	X =  362.589  mm,	Y =   -421.573  mm,	Z =   -258.355  mm,
	W =  90.000 deg,	P =   0.000 deg,	R =   90.000 deg
};
P[1425]{
   GP1:
	UF : 0, UT : 6,		CONFIG : 'N U T, 0, 0, 0',
	X =  364.293  mm,	Y =   -420.662  mm,	Z =   -257.910  mm,
	W =  90.000 deg,	P =   0.000 deg,	R =   90.000 deg
};
P[1426]{
   GP1:
	UF : 0, UT : 6,		CONFIG : 'N U T, 0, 0, 0',
	X =  365.269  mm,	Y =   -420.040  mm,	Z =   -258.263  mm,
	W =  90.000 deg,	P =   0.000 deg,	R =   90.000 deg
};
P[1427]{
   GP1:
	UF : 0, UT : 6,		CONFIG : 'N U T, 0, 0, 0',
	X =  366.692  mm,	Y =   -418.972  mm,	Z =   -258.264  mm,
	W =  90.000 deg,	P =   0.000 deg,	R =   90.000 deg
};
P[1428]{
   GP1:
	UF : 0, UT : 6,		CONFIG : 'N U T, 0, 0, 0',
	X =  367.410  mm,	Y =   -418.013  mm,	Z =   -258.141  mm,
	W =  90.000 deg,	P =   0.000 deg,	R =   90.000 deg
};
P[1429]{
   GP1:
	UF : 0, UT : 6,		CONFIG : 'N U T, 0, 0, 0',
	X =  367.867  mm,	Y =   -416.103  mm,	Z =   -258.050  mm,
	W =  90.000 deg,	P =   0.000 deg,	R =   90.000 deg
};
P[1430]{
   GP1:
	UF : 0, UT : 6,		CONFIG : 'N U T, 0, 0, 0',
	X =  366.496  mm,	Y =   -412.696  mm,	Z =   -258.023  mm,
	W =  90.000 deg,	P =   0.000 deg,	R =   90.000 deg
};
P[1431]{
   GP1:
	UF : 0, UT : 6,		CONFIG : 'N U T, 0, 0, 0',
	X =  365.953  mm,	Y =   -411.845  mm,	Z =   -258.338  mm,
	W =  90.000 deg,	P =   0.000 deg,	R =   90.000 deg
};
P[1432]{
   GP1:
	UF : 0, UT : 6,		CONFIG : 'N U T, 0, 0, 0',
	X =  365.463  mm,	Y =   -410.938  mm,	Z =   -258.135  mm,
	W =  90.000 deg,	P =   0.000 deg,	R =   90.000 deg
};
P[1433]{
   GP1:
	UF : 0, UT : 6,		CONFIG : 'N U T, 0, 0, 0',
	X =  364.194  mm,	Y =   -408.723  mm,	Z =   -258.077  mm,
	W =  90.000 deg,	P =   0.000 deg,	R =   90.000 deg
};
P[1434]{
   GP1:
	UF : 0, UT : 6,		CONFIG : 'N U T, 0, 0, 0',
	X =  363.608  mm,	Y =   -407.735  mm,	Z =   -258.173  mm,
	W =  90.000 deg,	P =   0.000 deg,	R =   90.000 deg
};
P[1435]{
   GP1:
	UF : 0, UT : 6,		CONFIG : 'N U T, 0, 0, 0',
	X =  363.116  mm,	Y =   -406.844  mm,	Z =   -258.027  mm,
	W =  90.000 deg,	P =   0.000 deg,	R =   90.000 deg
};
P[1436]{
   GP1:
	UF : 0, UT : 6,		CONFIG : 'N U T, 0, 0, 0',
	X =  362.751  mm,	Y =   -406.265  mm,	Z =   -258.222  mm,
	W =  90.000 deg,	P =   0.000 deg,	R =   90.000 deg
};
P[1437]{
   GP1:
	UF : 0, UT : 6,		CONFIG : 'N U T, 0, 0, 0',
	X =  362.005  mm,	Y =   -404.911  mm,	Z =   -257.998  mm,
	W =  90.000 deg,	P =   0.000 deg,	R =   90.000 deg
};
P[1438]{
   GP1:
	UF : 0, UT : 6,		CONFIG : 'N U T, 0, 0, 0',
	X =  361.348  mm,	Y =   -403.797  mm,	Z =   -258.091  mm,
	W =  90.000 deg,	P =   0.000 deg,	R =   90.000 deg
};
P[1439]{
   GP1:
	UF : 0, UT : 6,		CONFIG : 'N U T, 0, 0, 0',
	X =  360.844  mm,	Y =   -402.946  mm,	Z =   -258.162  mm,
	W =  90.000 deg,	P =   0.000 deg,	R =   90.000 deg
};
P[1440]{
   GP1:
	UF : 0, UT : 6,		CONFIG : 'N U T, 0, 0, 0',
	X =  359.010  mm,	Y =   -399.763  mm,	Z =   -258.140  mm,
	W =  90.000 deg,	P =   0.000 deg,	R =   90.000 deg
};
P[1441]{
   GP1:
	UF : 0, UT : 6,		CONFIG : 'N U T, 0, 0, 0',
	X =  358.114  mm,	Y =   -398.191  mm,	Z =   -258.065  mm,
	W =  90.000 deg,	P =   0.000 deg,	R =   90.000 deg
};
P[1442]{
   GP1:
	UF : 0, UT : 6,		CONFIG : 'N U T, 0, 0, 0',
	X =  357.785  mm,	Y =   -397.593  mm,	Z =   -257.963  mm,
	W =  90.000 deg,	P =   0.000 deg,	R =   90.000 deg
};
P[1443]{
   GP1:
	UF : 0, UT : 6,		CONFIG : 'N U T, 0, 0, 0',
	X =  356.865  mm,	Y =   -396.019  mm,	Z =   -258.034  mm,
	W =  90.000 deg,	P =   0.000 deg,	R =   90.000 deg
};
P[1444]{
   GP1:
	UF : 0, UT : 6,		CONFIG : 'N U T, 0, 0, 0',
	X =  355.938  mm,	Y =   -394.472  mm,	Z =   -258.241  mm,
	W =  90.000 deg,	P =   0.000 deg,	R =   90.000 deg
};
P[1445]{
   GP1:
	UF : 0, UT : 6,		CONFIG : 'N U T, 0, 0, 0',
	X =  355.370  mm,	Y =   -393.472  mm,	Z =   -258.186  mm,
	W =  90.000 deg,	P =   0.000 deg,	R =   90.000 deg
};
P[1446]{
   GP1:
	UF : 0, UT : 6,		CONFIG : 'N U T, 0, 0, 0',
	X =  354.801  mm,	Y =   -392.444  mm,	Z =   -258.035  mm,
	W =  90.000 deg,	P =   0.000 deg,	R =   90.000 deg
};
P[1447]{
   GP1:
	UF : 0, UT : 6,		CONFIG : 'N U T, 0, 0, 0',
	X =  353.910  mm,	Y =   -390.927  mm,	Z =   -258.124  mm,
	W =  90.000 deg,	P =   0.000 deg,	R =   90.000 deg
};
P[1448]{
   GP1:
	UF : 0, UT : 6,		CONFIG : 'N U T, 0, 0, 0',
	X =  353.521  mm,	Y =   -390.306  mm,	Z =   -258.315  mm,
	W =  90.000 deg,	P =   0.000 deg,	R =   90.000 deg
};
P[1449]{
   GP1:
	UF : 0, UT : 6,		CONFIG : 'N U T, 0, 0, 0',
	X =  353.090  mm,	Y =   -389.550  mm,	Z =   -258.278  mm,
	W =  90.000 deg,	P =   0.000 deg,	R =   90.000 deg
};
P[1450]{
   GP1:
	UF : 0, UT : 6,		CONFIG : 'N U T, 0, 0, 0',
	X =  352.400  mm,	Y =   -388.329  mm,	Z =   -258.184  mm,
	W =  90.000 deg,	P =   0.000 deg,	R =   90.000 deg
};
P[1451]{
   GP1:
	UF : 0, UT : 6,		CONFIG : 'N U T, 0, 0, 0',
	X =  351.577  mm,	Y =   -386.900  mm,	Z =   -258.175  mm,
	W =  90.000 deg,	P =   0.000 deg,	R =   90.000 deg
};
P[1452]{
   GP1:
	UF : 0, UT : 6,		CONFIG : 'N U T, 0, 0, 0',
	X =  350.872  mm,	Y =   -385.686  mm,	Z =   -258.199  mm,
	W =  90.000 deg,	P =   0.000 deg,	R =   90.000 deg
};
P[1453]{
   GP1:
	UF : 0, UT : 6,		CONFIG : 'N U T, 0, 0, 0',
	X =  350.224  mm,	Y =   -384.589  mm,	Z =   -258.293  mm,
	W =  90.000 deg,	P =   0.000 deg,	R =   90.000 deg
};
P[1454]{
   GP1:
	UF : 0, UT : 6,		CONFIG : 'N U T, 0, 0, 0',
	X =  349.367  mm,	Y =   -383.063  mm,	Z =   -258.140  mm,
	W =  90.000 deg,	P =   0.000 deg,	R =   90.000 deg
};
P[1455]{
   GP1:
	UF : 0, UT : 6,		CONFIG : 'N U T, 0, 0, 0',
	X =  347.541  mm,	Y =   -379.863  mm,	Z =   -258.004  mm,
	W =  90.000 deg,	P =   0.000 deg,	R =   90.000 deg
};
P[1456]{
   GP1:
	UF : 0, UT : 6,		CONFIG : 'N U T, 0, 0, 0',
	X =  346.802  mm,	Y =   -378.617  mm,	Z =   -258.126  mm,
	W =  90.000 deg,	P =   0.000 deg,	R =   90.000 deg
};
P[1457]{
   GP1:
	UF : 0, UT : 6,		CONFIG : 'N U T, 0, 0, 0',
	X =  346.157  mm,	Y =   -377.558  mm,	Z =   -258.332  mm,
	W =  90.000 deg,	P =   0.000 deg,	R =   90.000 deg
};
P[1458]{
   GP1:
	UF : 0, UT : 6,		CONFIG : 'N U T, 0, 0, 0',
	X =  343.463  mm,	Y =   -372.896  mm,	Z =   -258.352  mm,
	W =  90.000 deg,	P =   0.000 deg,	R =   90.000 deg
};
P[1459]{
   GP1:
	UF : 0, UT : 6,		CONFIG : 'N U T, 0, 0, 0',
	X =  341.709  mm,	Y =   -369.779  mm,	Z =   -258.066  mm,
	W =  90.000 deg,	P =   0.000 deg,	R =   90.000 deg
};
P[1460]{
   GP1:
	UF : 0, UT : 6,		CONFIG : 'N U T, 0, 0, 0',
	X =  341.083  mm,	Y =   -368.700  mm,	Z =   -258.086  mm,
	W =  90.000 deg,	P =   0.000 deg,	R =   90.000 deg
};
P[1461]{
   GP1:
	UF : 0, UT : 6,		CONFIG : 'N U T, 0, 0, 0',
	X =  340.436  mm,	Y =   -367.555  mm,	Z =   -257.993  mm,
	W =  90.000 deg,	P =   0.000 deg,	R =   90.000 deg
};
P[1462]{
   GP1:
	UF : 0, UT : 6,		CONFIG : 'N U T, 0, 0, 0',
	X =  339.501  mm,	Y =   -366.020  mm,	Z =   -258.301  mm,
	W =  90.000 deg,	P =   0.000 deg,	R =   90.000 deg
};
P[1463]{
   GP1:
	UF : 0, UT : 6,		CONFIG : 'N U T, 0, 0, 0',
	X =  337.784  mm,	Y =   -363.056  mm,	Z =   -258.335  mm,
	W =  90.000 deg,	P =   0.000 deg,	R =   90.000 deg
};
P[1464]{
   GP1:
	UF : 0, UT : 6,		CONFIG : 'N U T, 0, 0, 0',
	X =  334.814  mm,	Y =   -357.912  mm,	Z =   -258.333  mm,
	W =  90.000 deg,	P =   0.000 deg,	R =   90.000 deg
};
P[1465]{
   GP1:
	UF : 0, UT : 6,		CONFIG : 'N U T, 0, 0, 0',
	X =  334.136  mm,	Y =   -356.713  mm,	Z =   -258.245  mm,
	W =  90.000 deg,	P =   0.000 deg,	R =   90.000 deg
};
P[1466]{
   GP1:
	UF : 0, UT : 6,		CONFIG : 'N U T, 0, 0, 0',
	X =  333.471  mm,	Y =   -355.599  mm,	Z =   -258.374  mm,
	W =  90.000 deg,	P =   0.000 deg,	R =   90.000 deg
};
P[1467]{
   GP1:
	UF : 0, UT : 6,		CONFIG : 'N U T, 0, 0, 0',
	X =  332.196  mm,	Y =   -353.372  mm,	Z =   -258.310  mm,
	W =  90.000 deg,	P =   0.000 deg,	R =   90.000 deg
};
P[1468]{
   GP1:
	UF : 0, UT : 6,		CONFIG : 'N U T, 0, 0, 0',
	X =  331.933  mm,	Y =   -352.844  mm,	Z =   -258.055  mm,
	W =  90.000 deg,	P =   0.000 deg,	R =   90.000 deg
};
P[1469]{
   GP1:
	UF : 0, UT : 6,		CONFIG : 'N U T, 0, 0, 0',
	X =  329.978  mm,	Y =   -349.493  mm,	Z =   -258.179  mm,
	W =  90.000 deg,	P =   0.000 deg,	R =   90.000 deg
};
P[1470]{
   GP1:
	UF : 0, UT : 6,		CONFIG : 'N U T, 0, 0, 0',
	X =  328.764  mm,	Y =   -347.342  mm,	Z =   -258.012  mm,
	W =  90.000 deg,	P =   0.000 deg,	R =   90.000 deg
};
P[1471]{
   GP1:
	UF : 0, UT : 6,		CONFIG : 'N U T, 0, 0, 0',
	X =  327.979  mm,	Y =   -346.076  mm,	Z =   -258.343  mm,
	W =  90.000 deg,	P =   0.000 deg,	R =   90.000 deg
};
P[1472]{
   GP1:
	UF : 0, UT : 6,		CONFIG : 'N U T, 0, 0, 0',
	X =  327.666  mm,	Y =   -345.482  mm,	Z =   -258.155  mm,
	W =  90.000 deg,	P =   0.000 deg,	R =   90.000 deg
};
P[1473]{
   GP1:
	UF : 0, UT : 6,		CONFIG : 'N U T, 0, 0, 0',
	X =  327.287  mm,	Y =   -344.772  mm,	Z =   -257.960  mm,
	W =  90.000 deg,	P =   0.000 deg,	R =   90.000 deg
};
P[1474]{
   GP1:
	UF : 0, UT : 6,		CONFIG : 'N U T, 0, 0, 0',
	X =  326.614  mm,	Y =   -343.677  mm,	Z =   -258.215  mm,
	W =  90.000 deg,	P =   0.000 deg,	R =   90.000 deg
};
P[1475]{
   GP1:
	UF : 0, UT : 6,		CONFIG : 'N U T, 0, 0, 0',
	X =  325.548  mm,	Y =   -341.865  mm,	Z =   -258.335  mm,
	W =  90.000 deg,	P =   0.000 deg,	R =   90.000 deg
};
P[1476]{
   GP1:
	UF : 0, UT : 6,		CONFIG : 'N U T, 0, 0, 0',
	X =  323.271  mm,	Y =   -337.797  mm,	Z =   -257.899  mm,
	W =  90.000 deg,	P =   0.000 deg,	R =   90.000 deg
};
P[1477]{
   GP1:
	UF : 0, UT : 6,		CONFIG : 'N U T, 0, 0, 0',
	X =  322.557  mm,	Y =   -336.645  mm,	Z =   -258.194  mm,
	W =  90.000 deg,	P =   0.000 deg,	R =   90.000 deg
};
P[1478]{
   GP1:
	UF : 0, UT : 6,		CONFIG : 'N U T, 0, 0, 0',
	X =  322.106  mm,	Y =   -335.851  mm,	Z =   -258.147  mm,
	W =  90.000 deg,	P =   0.000 deg,	R =   90.000 deg
};
P[1479]{
   GP1:
	UF : 0, UT : 6,		CONFIG : 'N U T, 0, 0, 0',
	X =  321.016  mm,	Y =   -334.011  mm,	Z =   -258.319  mm,
	W =  90.000 deg,	P =   0.000 deg,	R =   90.000 deg
};
P[1480]{
   GP1:
	UF : 0, UT : 6,		CONFIG : 'N U T, 0, 0, 0',
	X =  320.706  mm,	Y =   -333.426  mm,	Z =   -258.143  mm,
	W =  90.000 deg,	P =   0.000 deg,	R =   90.000 deg
};
P[1481]{
   GP1:
	UF : 0, UT : 6,		CONFIG : 'N U T, 0, 0, 0',
	X =  319.386  mm,	Y =   -331.178  mm,	Z =   -258.283  mm,
	W =  90.000 deg,	P =   0.000 deg,	R =   90.000 deg
};
P[1482]{
   GP1:
	UF : 0, UT : 6,		CONFIG : 'N U T, 0, 0, 0',
	X =  318.670  mm,	Y =   -329.897  mm,	Z =   -258.143  mm,
	W =  90.000 deg,	P =   0.000 deg,	R =   90.000 deg
};
P[1483]{
   GP1:
	UF : 0, UT : 6,		CONFIG : 'N U T, 0, 0, 0',
	X =  318.040  mm,	Y =   -328.736  mm,	Z =   -257.885  mm,
	W =  90.000 deg,	P =   0.000 deg,	R =   90.000 deg
};
P[1484]{
   GP1:
	UF : 0, UT : 6,		CONFIG : 'N U T, 0, 0, 0',
	X =  316.598  mm,	Y =   -326.306  mm,	Z =   -258.135  mm,
	W =  90.000 deg,	P =   0.000 deg,	R =   90.000 deg
};
P[1485]{
   GP1:
	UF : 0, UT : 6,		CONFIG : 'N U T, 0, 0, 0',
	X =  316.051  mm,	Y =   -325.402  mm,	Z =   -258.288  mm,
	W =  90.000 deg,	P =   0.000 deg,	R =   90.000 deg
};
P[1486]{
   GP1:
	UF : 0, UT : 6,		CONFIG : 'N U T, 0, 0, 0',
	X =  313.801  mm,	Y =   -321.453  mm,	Z =   -258.102  mm,
	W =  90.000 deg,	P =   0.000 deg,	R =   90.000 deg
};
P[1487]{
   GP1:
	UF : 0, UT : 6,		CONFIG : 'N U T, 0, 0, 0',
	X =  313.176  mm,	Y =   -320.327  mm,	Z =   -257.941  mm,
	W =  90.000 deg,	P =   0.000 deg,	R =   90.000 deg
};
P[1488]{
   GP1:
	UF : 0, UT : 6,		CONFIG : 'N U T, 0, 0, 0',
	X =  312.368  mm,	Y =   -318.999  mm,	Z =   -258.195  mm,
	W =  90.000 deg,	P =   0.000 deg,	R =   90.000 deg
};
P[1489]{
   GP1:
	UF : 0, UT : 6,		CONFIG : 'N U T, 0, 0, 0',
	X =  311.565  mm,	Y =   -317.609  mm,	Z =   -258.199  mm,
	W =  90.000 deg,	P =   0.000 deg,	R =   90.000 deg
};
P[1490]{
   GP1:
	UF : 0, UT : 6,		CONFIG : 'N U T, 0, 0, 0',
	X =  310.607  mm,	Y =   -315.929  mm,	Z =   -258.128  mm,
	W =  90.000 deg,	P =   0.000 deg,	R =   90.000 deg
};
P[1491]{
   GP1:
	UF : 0, UT : 6,		CONFIG : 'N U T, 0, 0, 0',
	X =  310.120  mm,	Y =   -315.110  mm,	Z =   -258.211  mm,
	W =  90.000 deg,	P =   0.000 deg,	R =   90.000 deg
};
P[1492]{
   GP1:
	UF : 0, UT : 6,		CONFIG : 'N U T, 0, 0, 0',
	X =  309.509  mm,	Y =   -314.037  mm,	Z =   -258.158  mm,
	W =  90.000 deg,	P =   0.000 deg,	R =   90.000 deg
};
P[1493]{
   GP1:
	UF : 0, UT : 6,		CONFIG : 'N U T, 0, 0, 0',
	X =  309.119  mm,	Y =   -313.374  mm,	Z =   -258.209  mm,
	W =  90.000 deg,	P =   0.000 deg,	R =   90.000 deg
};
P[1494]{
   GP1:
	UF : 0, UT : 6,		CONFIG : 'N U T, 0, 0, 0',
	X =  308.501  mm,	Y =   -312.233  mm,	Z =   -257.955  mm,
	W =  90.000 deg,	P =   0.000 deg,	R =   90.000 deg
};
P[1495]{
   GP1:
	UF : 0, UT : 6,		CONFIG : 'N U T, 0, 0, 0',
	X =  307.294  mm,	Y =   -310.255  mm,	Z =   -258.354  mm,
	W =  90.000 deg,	P =   0.000 deg,	R =   90.000 deg
};
P[1496]{
   GP1:
	UF : 0, UT : 6,		CONFIG : 'N U T, 0, 0, 0',
	X =  306.652  mm,	Y =   -309.123  mm,	Z =   -258.287  mm,
	W =  90.000 deg,	P =   0.000 deg,	R =   90.000 deg
};
P[1497]{
   GP1:
	UF : 0, UT : 6,		CONFIG : 'N U T, 0, 0, 0',
	X =  305.969  mm,	Y =   -307.954  mm,	Z =   -258.332  mm,
	W =  90.000 deg,	P =   0.000 deg,	R =   90.000 deg
};
P[1498]{
   GP1:
	UF : 0, UT : 6,		CONFIG : 'N U T, 0, 0, 0',
	X =  305.470  mm,	Y =   -306.980  mm,	Z =   -257.938  mm,
	W =  90.000 deg,	P =   0.000 deg,	R =   90.000 deg
};
P[1499]{
   GP1:
	UF : 0, UT : 6,		CONFIG : 'N U T, 0, 0, 0',
	X =  304.036  mm,	Y =   -304.589  mm,	Z =   -258.275  mm,
	W =  90.000 deg,	P =   0.000 deg,	R =   90.000 deg
};
P[1500]{
   GP1:
	UF : 0, UT : 6,		CONFIG : 'N U T, 0, 0, 0',
	X =  303.387  mm,	Y =   -303.450  mm,	Z =   -258.220  mm,
	W =  90.000 deg,	P =   0.000 deg,	R =   90.000 deg
};
P[1501]{
   GP1:
	UF : 0, UT : 6,		CONFIG : 'N U T, 0, 0, 0',
	X =  302.854  mm,	Y =   -302.518  mm,	Z =   -258.187  mm,
	W =  90.000 deg,	P =   0.000 deg,	R =   90.000 deg
};
P[1502]{
   GP1:
	UF : 0, UT : 6,		CONFIG : 'N U T, 0, 0, 0',
	X =  301.892  mm,	Y =   -300.793  mm,	Z =   -257.974  mm,
	W =  90.000 deg,	P =   0.000 deg,	R =   90.000 deg
};
P[1503]{
   GP1:
	UF : 0, UT : 6,		CONFIG : 'N U T, 0, 0, 0',
	X =  301.154  mm,	Y =   -299.524  mm,	Z =   -258.006  mm,
	W =  90.000 deg,	P =   0.000 deg,	R =   90.000 deg
};
P[1504]{
   GP1:
	UF : 0, UT : 6,		CONFIG : 'N U T, 0, 0, 0',
	X =  300.062  mm,	Y =   -297.699  mm,	Z =   -258.244  mm,
	W =  90.000 deg,	P =   0.000 deg,	R =   90.000 deg
};
P[1505]{
   GP1:
	UF : 0, UT : 6,		CONFIG : 'N U T, 0, 0, 0',
	X =  299.663  mm,	Y =   -296.945  mm,	Z =   -258.024  mm,
	W =  90.000 deg,	P =   0.000 deg,	R =   90.000 deg
};
P[1506]{
   GP1:
	UF : 0, UT : 6,		CONFIG : 'N U T, 0, 0, 0',
	X =  299.022  mm,	Y =   -295.910  mm,	Z =   -258.287  mm,
	W =  90.000 deg,	P =   0.000 deg,	R =   90.000 deg
};
P[1507]{
   GP1:
	UF : 0, UT : 6,		CONFIG : 'N U T, 0, 0, 0',
	X =  298.421  mm,	Y =   -294.812  mm,	Z =   -258.079  mm,
	W =  90.000 deg,	P =   0.000 deg,	R =   90.000 deg
};
P[1508]{
   GP1:
	UF : 0, UT : 6,		CONFIG : 'N U T, 0, 0, 0',
	X =  297.989  mm,	Y =   -294.136  mm,	Z =   -258.340  mm,
	W =  90.000 deg,	P =   0.000 deg,	R =   90.000 deg
};
P[1509]{
   GP1:
	UF : 0, UT : 6,		CONFIG : 'N U T, 0, 0, 0',
	X =  297.665  mm,	Y =   -293.480  mm,	Z =   -258.000  mm,
	W =  90.000 deg,	P =   0.000 deg,	R =   90.000 deg
};
P[1510]{
   GP1:
	UF : 0, UT : 6,		CONFIG : 'N U T, 0, 0, 0',
	X =  297.270  mm,	Y =   -292.767  mm,	Z =   -257.901  mm,
	W =  90.000 deg,	P =   0.000 deg,	R =   90.000 deg
};
P[1511]{
   GP1:
	UF : 0, UT : 6,		CONFIG : 'N U T, 0, 0, 0',
	X =  296.800  mm,	Y =   -291.997  mm,	Z =   -258.058  mm,
	W =  90.000 deg,	P =   0.000 deg,	R =   90.000 deg
};
P[1512]{
   GP1:
	UF : 0, UT : 6,		CONFIG : 'N U T, 0, 0, 0',
	X =  296.307  mm,	Y =   -291.107  mm,	Z =   -257.931  mm,
	W =  90.000 deg,	P =   0.000 deg,	R =   90.000 deg
};
P[1513]{
   GP1:
	UF : 0, UT : 6,		CONFIG : 'N U T, 0, 0, 0',
	X =  295.808  mm,	Y =   -290.360  mm,	Z =   -258.343  mm,
	W =  90.000 deg,	P =   0.000 deg,	R =   90.000 deg
};
P[1514]{
   GP1:
	UF : 0, UT : 6,		CONFIG : 'N U T, 0, 0, 0',
	X =  294.775  mm,	Y =   -288.532  mm,	Z =   -258.203  mm,
	W =  90.000 deg,	P =   0.000 deg,	R =   90.000 deg
};
P[1515]{
   GP1:
	UF : 0, UT : 6,		CONFIG : 'N U T, 0, 0, 0',
	X =  293.528  mm,	Y =   -286.314  mm,	Z =   -258.001  mm,
	W =  90.000 deg,	P =   0.000 deg,	R =   90.000 deg
};
P[1516]{
   GP1:
	UF : 0, UT : 6,		CONFIG : 'N U T, 0, 0, 0',
	X =  292.967  mm,	Y =   -285.425  mm,	Z =   -258.292  mm,
	W =  90.000 deg,	P =   0.000 deg,	R =   90.000 deg
};
P[1517]{
   GP1:
	UF : 0, UT : 6,		CONFIG : 'N U T, 0, 0, 0',
	X =  292.494  mm,	Y =   -284.556  mm,	Z =   -258.111  mm,
	W =  90.000 deg,	P =   0.000 deg,	R =   90.000 deg
};
P[1518]{
   GP1:
	UF : 0, UT : 6,		CONFIG : 'N U T, 0, 0, 0',
	X =  291.586  mm,	Y =   -283.048  mm,	Z =   -258.349  mm,
	W =  90.000 deg,	P =   0.000 deg,	R =   90.000 deg
};
P[1519]{
   GP1:
	UF : 0, UT : 6,		CONFIG : 'N U T, 0, 0, 0',
	X =  290.775  mm,	Y =   -281.622  mm,	Z =   -258.268  mm,
	W =  90.000 deg,	P =   0.000 deg,	R =   90.000 deg
};
P[1520]{
   GP1:
	UF : 0, UT : 6,		CONFIG : 'N U T, 0, 0, 0',
	X =  290.106  mm,	Y =   -280.403  mm,	Z =   -258.058  mm,
	W =  90.000 deg,	P =   0.000 deg,	R =   90.000 deg
};
P[1521]{
   GP1:
	UF : 0, UT : 6,		CONFIG : 'N U T, 0, 0, 0',
	X =  289.351  mm,	Y =   -279.154  mm,	Z =   -258.263  mm,
	W =  90.000 deg,	P =   0.000 deg,	R =   90.000 deg
};
P[1522]{
   GP1:
	UF : 0, UT : 6,		CONFIG : 'N U T, 0, 0, 0',
	X =  288.798  mm,	Y =   -278.197  mm,	Z =   -258.268  mm,
	W =  90.000 deg,	P =   0.000 deg,	R =   90.000 deg
};
P[1523]{
   GP1:
	UF : 0, UT : 6,		CONFIG : 'N U T, 0, 0, 0',
	X =  287.513  mm,	Y =   -275.976  mm,	Z =   -258.286  mm,
	W =  90.000 deg,	P =   0.000 deg,	R =   90.000 deg
};
P[1524]{
   GP1:
	UF : 0, UT : 6,		CONFIG : 'N U T, 0, 0, 0',
	X =  286.825  mm,	Y =   -274.773  mm,	Z =   -258.248  mm,
	W =  90.000 deg,	P =   0.000 deg,	R =   90.000 deg
};
P[1525]{
   GP1:
	UF : 0, UT : 6,		CONFIG : 'N U T, 0, 0, 0',
	X =  285.617  mm,	Y =   -272.667  mm,	Z =   -258.193  mm,
	W =  90.000 deg,	P =   0.000 deg,	R =   90.000 deg
};
P[1526]{
   GP1:
	UF : 0, UT : 6,		CONFIG : 'N U T, 0, 0, 0',
	X =  285.296  mm,	Y =   -272.065  mm,	Z =   -258.029  mm,
	W =  90.000 deg,	P =   0.000 deg,	R =   90.000 deg
};
P[1527]{
   GP1:
	UF : 0, UT : 6,		CONFIG : 'N U T, 0, 0, 0',
	X =  283.770  mm,	Y =   -269.457  mm,	Z =   -258.156  mm,
	W =  90.000 deg,	P =   0.000 deg,	R =   90.000 deg
};
P[1528]{
   GP1:
	UF : 0, UT : 6,		CONFIG : 'N U T, 0, 0, 0',
	X =  283.265  mm,	Y =   -268.628  mm,	Z =   -258.321  mm,
	W =  90.000 deg,	P =   0.000 deg,	R =   90.000 deg
};
P[1529]{
   GP1:
	UF : 0, UT : 6,		CONFIG : 'N U T, 0, 0, 0',
	X =  282.607  mm,	Y =   -267.473  mm,	Z =   -258.262  mm,
	W =  90.000 deg,	P =   0.000 deg,	R =   90.000 deg
};
P[1530]{
   GP1:
	UF : 0, UT : 6,		CONFIG : 'N U T, 0, 0, 0',
	X =  282.017  mm,	Y =   -266.418  mm,	Z =   -258.150  mm,
	W =  90.000 deg,	P =   0.000 deg,	R =   90.000 deg
};
P[1531]{
   GP1:
	UF : 0, UT : 6,		CONFIG : 'N U T, 0, 0, 0',
	X =  281.454  mm,	Y =   -265.451  mm,	Z =   -258.172  mm,
	W =  90.000 deg,	P =   0.000 deg,	R =   90.000 deg
};
P[1532]{
   GP1:
	UF : 0, UT : 6,		CONFIG : 'N U T, 0, 0, 0',
	X =  280.944  mm,	Y =   -264.578  mm,	Z =   -258.206  mm,
	W =  90.000 deg,	P =   0.000 deg,	R =   90.000 deg
};
P[1533]{
   GP1:
	UF : 0, UT : 6,		CONFIG : 'N U T, 0, 0, 0',
	X =  280.627  mm,	Y =   -263.992  mm,	Z =   -258.071  mm,
	W =  90.000 deg,	P =   0.000 deg,	R =   90.000 deg
};
P[1534]{
   GP1:
	UF : 0, UT : 6,		CONFIG : 'N U T, 0, 0, 0',
	X =  279.920  mm,	Y =   -262.842  mm,	Z =   -258.346  mm,
	W =  90.000 deg,	P =   0.000 deg,	R =   90.000 deg
};
P[1535]{
   GP1:
	UF : 0, UT : 6,		CONFIG : 'N U T, 0, 0, 0',
	X =  279.313  mm,	Y =   -261.717  mm,	Z =   -258.081  mm,
	W =  90.000 deg,	P =   0.000 deg,	R =   90.000 deg
};
P[1536]{
   GP1:
	UF : 0, UT : 6,		CONFIG : 'N U T, 0, 0, 0',
	X =  278.629  mm,	Y =   -260.587  mm,	Z =   -258.274  mm,
	W =  90.000 deg,	P =   0.000 deg,	R =   90.000 deg
};
P[1537]{
   GP1:
	UF : 0, UT : 6,		CONFIG : 'N U T, 0, 0, 0',
	X =  277.377  mm,	Y =   -258.401  mm,	Z =   -258.210  mm,
	W =  90.000 deg,	P =   0.000 deg,	R =   90.000 deg
};
P[1538]{
   GP1:
	UF : 0, UT : 6,		CONFIG : 'N U T, 0, 0, 0',
	X =  276.891  mm,	Y =   -257.580  mm,	Z =   -258.287  mm,
	W =  90.000 deg,	P =   0.000 deg,	R =   90.000 deg
};
P[1539]{
   GP1:
	UF : 0, UT : 6,		CONFIG : 'N U T, 0, 0, 0',
	X =  276.404  mm,	Y =   -256.709  mm,	Z =   -258.189  mm,
	W =  90.000 deg,	P =   0.000 deg,	R =   90.000 deg
};
P[1540]{
   GP1:
	UF : 0, UT : 6,		CONFIG : 'N U T, 0, 0, 0',
	X =  275.581  mm,	Y =   -255.216  mm,	Z =   -257.949  mm,
	W =  90.000 deg,	P =   0.000 deg,	R =   90.000 deg
};
P[1541]{
   GP1:
	UF : 0, UT : 6,		CONFIG : 'N U T, 0, 0, 0',
	X =  275.157  mm,	Y =   -254.541  mm,	Z =   -258.157  mm,
	W =  90.000 deg,	P =   0.000 deg,	R =   90.000 deg
};
P[1542]{
   GP1:
	UF : 0, UT : 6,		CONFIG : 'N U T, 0, 0, 0',
	X =  274.353  mm,	Y =   -253.114  mm,	Z =   -258.035  mm,
	W =  90.000 deg,	P =   0.000 deg,	R =   90.000 deg
};
P[1543]{
   GP1:
	UF : 0, UT : 6,		CONFIG : 'N U T, 0, 0, 0',
	X =  273.454  mm,	Y =   -251.617  mm,	Z =   -258.248  mm,
	W =  90.000 deg,	P =   0.000 deg,	R =   90.000 deg
};
P[1544]{
   GP1:
	UF : 0, UT : 6,		CONFIG : 'N U T, 0, 0, 0',
	X =  273.055  mm,	Y =   -250.939  mm,	Z =   -258.289  mm,
	W =  90.000 deg,	P =   0.000 deg,	R =   90.000 deg
};
P[1545]{
   GP1:
	UF : 0, UT : 6,		CONFIG : 'N U T, 0, 0, 0',
	X =  272.617  mm,	Y =   -250.161  mm,	Z =   -258.227  mm,
	W =  90.000 deg,	P =   0.000 deg,	R =   90.000 deg
};
P[1546]{
   GP1:
	UF : 0, UT : 6,		CONFIG : 'N U T, 0, 0, 0',
	X =  272.242  mm,	Y =   -249.508  mm,	Z =   -258.214  mm,
	W =  90.000 deg,	P =   0.000 deg,	R =   90.000 deg
};
P[1547]{
   GP1:
	UF : 0, UT : 6,		CONFIG : 'N U T, 0, 0, 0',
	X =  271.714  mm,	Y =   -248.613  mm,	Z =   -258.278  mm,
	W =  90.000 deg,	P =   0.000 deg,	R =   90.000 deg
};
P[1548]{
   GP1:
	UF : 0, UT : 6,		CONFIG : 'N U T, 0, 0, 0',
	X =  271.157  mm,	Y =   -247.674  mm,	Z =   -258.369  mm,
	W =  90.000 deg,	P =   0.000 deg,	R =   90.000 deg
};
P[1549]{
   GP1:
	UF : 0, UT : 6,		CONFIG : 'N U T, 0, 0, 0',
	X =  270.028  mm,	Y =   -245.625  mm,	Z =   -258.039  mm,
	W =  90.000 deg,	P =   0.000 deg,	R =   90.000 deg
};
P[1550]{
   GP1:
	UF : 0, UT : 6,		CONFIG : 'N U T, 0, 0, 0',
	X =  269.417  mm,	Y =   -244.548  mm,	Z =   -257.979  mm,
	W =  90.000 deg,	P =   0.000 deg,	R =   90.000 deg
};
P[1551]{
   GP1:
	UF : 0, UT : 6,		CONFIG : 'N U T, 0, 0, 0',
	X =  269.071  mm,	Y =   -244.040  mm,	Z =   -258.300  mm,
	W =  90.000 deg,	P =   0.000 deg,	R =   90.000 deg
};
P[1552]{
   GP1:
	UF : 0, UT : 6,		CONFIG : 'N U T, 0, 0, 0',
	X =  268.630  mm,	Y =   -243.256  mm,	Z =   -258.229  mm,
	W =  90.000 deg,	P =   0.000 deg,	R =   90.000 deg
};
P[1553]{
   GP1:
	UF : 0, UT : 6,		CONFIG : 'N U T, 0, 0, 0',
	X =  268.236  mm,	Y =   -242.610  mm,	Z =   -258.354  mm,
	W =  90.000 deg,	P =   0.000 deg,	R =   90.000 deg
};
P[1554]{
   GP1:
	UF : 0, UT : 6,		CONFIG : 'N U T, 0, 0, 0',
	X =  267.602  mm,	Y =   -241.484  mm,	Z =   -258.249  mm,
	W =  90.000 deg,	P =   0.000 deg,	R =   90.000 deg
};
P[1555]{
   GP1:
	UF : 0, UT : 6,		CONFIG : 'N U T, 0, 0, 0',
	X =  267.013  mm,	Y =   -240.456  mm,	Z =   -258.227  mm,
	W =  90.000 deg,	P =   0.000 deg,	R =   90.000 deg
};
P[1556]{
   GP1:
	UF : 0, UT : 6,		CONFIG : 'N U T, 0, 0, 0',
	X =  266.709  mm,	Y =   -239.844  mm,	Z =   -257.926  mm,
	W =  90.000 deg,	P =   0.000 deg,	R =   90.000 deg
};
P[1557]{
   GP1:
	UF : 0, UT : 6,		CONFIG : 'N U T, 0, 0, 0',
	X =  265.685  mm,	Y =   -238.177  mm,	Z =   -258.304  mm,
	W =  90.000 deg,	P =   0.000 deg,	R =   90.000 deg
};
P[1558]{
   GP1:
	UF : 0, UT : 6,		CONFIG : 'N U T, 0, 0, 0',
	X =  265.285  mm,	Y =   -237.411  mm,	Z =   -258.045  mm,
	W =  90.000 deg,	P =   0.000 deg,	R =   90.000 deg
};
P[1559]{
   GP1:
	UF : 0, UT : 6,		CONFIG : 'N U T, 0, 0, 0',
	X =  264.036  mm,	Y =   -235.228  mm,	Z =   -257.971  mm,
	W =  90.000 deg,	P =   0.000 deg,	R =   90.000 deg
};
P[1560]{
   GP1:
	UF : 0, UT : 6,		CONFIG : 'N U T, 0, 0, 0',
	X =  263.401  mm,	Y =   -234.143  mm,	Z =   -258.022  mm,
	W =  90.000 deg,	P =   0.000 deg,	R =   90.000 deg
};
P[1561]{
   GP1:
	UF : 0, UT : 6,		CONFIG : 'N U T, 0, 0, 0',
	X =  263.040  mm,	Y =   -233.616  mm,	Z =   -258.374  mm,
	W =  90.000 deg,	P =   0.000 deg,	R =   90.000 deg
};
P[1562]{
   GP1:
	UF : 0, UT : 6,		CONFIG : 'N U T, 0, 0, 0',
	X =  261.110  mm,	Y =   -230.213  mm,	Z =   -258.159  mm,
	W =  90.000 deg,	P =   0.000 deg,	R =   90.000 deg
};
P[1563]{
   GP1:
	UF : 0, UT : 6,		CONFIG : 'N U T, 0, 0, 0',
	X =  260.645  mm,	Y =   -229.352  mm,	Z =   -257.957  mm,
	W =  90.000 deg,	P =   0.000 deg,	R =   90.000 deg
};
P[1564]{
   GP1:
	UF : 0, UT : 6,		CONFIG : 'N U T, 0, 0, 0',
	X =  260.138  mm,	Y =   -228.575  mm,	Z =   -258.322  mm,
	W =  90.000 deg,	P =   0.000 deg,	R =   90.000 deg
};
P[1565]{
   GP1:
	UF : 0, UT : 6,		CONFIG : 'N U T, 0, 0, 0',
	X =  259.630  mm,	Y =   -227.600  mm,	Z =   -257.980  mm,
	W =  90.000 deg,	P =   0.000 deg,	R =   90.000 deg
};
P[1566]{
   GP1:
	UF : 0, UT : 6,		CONFIG : 'N U T, 0, 0, 0',
	X =  259.011  mm,	Y =   -226.599  mm,	Z =   -258.234  mm,
	W =  90.000 deg,	P =   0.000 deg,	R =   90.000 deg
};
P[1567]{
   GP1:
	UF : 0, UT : 6,		CONFIG : 'N U T, 0, 0, 0',
	X =  257.821  mm,	Y =   -224.493  mm,	Z =   -258.071  mm,
	W =  90.000 deg,	P =   0.000 deg,	R =   90.000 deg
};
P[1568]{
   GP1:
	UF : 0, UT : 6,		CONFIG : 'N U T, 0, 0, 0',
	X =  256.302  mm,	Y =   -221.912  mm,	Z =   -258.253  mm,
	W =  90.000 deg,	P =   0.000 deg,	R =   90.000 deg
};
P[1569]{
   GP1:
	UF : 0, UT : 6,		CONFIG : 'N U T, 0, 0, 0',
	X =  255.604  mm,	Y =   -220.725  mm,	Z =   -258.333  mm,
	W =  90.000 deg,	P =   0.000 deg,	R =   90.000 deg
};
P[1570]{
   GP1:
	UF : 0, UT : 6,		CONFIG : 'N U T, 0, 0, 0',
	X =  255.085  mm,	Y =   -219.828  mm,	Z =   -258.337  mm,
	W =  90.000 deg,	P =   0.000 deg,	R =   90.000 deg
};
P[1571]{
   GP1:
	UF : 0, UT : 6,		CONFIG : 'N U T, 0, 0, 0',
	X =  254.679  mm,	Y =   -219.158  mm,	Z =   -258.361  mm,
	W =  90.000 deg,	P =   0.000 deg,	R =   90.000 deg
};
P[1572]{
   GP1:
	UF : 0, UT : 6,		CONFIG : 'N U T, 0, 0, 0',
	X =  253.477  mm,	Y =   -217.834  mm,	Z =   -258.012  mm,
	W =  90.000 deg,	P =   0.000 deg,	R =   90.000 deg
};
P[1573]{
   GP1:
	UF : 0, UT : 6,		CONFIG : 'N U T, 0, 0, 0',
	X =  252.099  mm,	Y =   -217.289  mm,	Z =   -258.202  mm,
	W =  90.000 deg,	P =   0.000 deg,	R =   90.000 deg
};
P[1574]{
   GP1:
	UF : 0, UT : 6,		CONFIG : 'N U T, 0, 0, 0',
	X =  250.979  mm,	Y =   -217.201  mm,	Z =   -258.331  mm,
	W =  90.000 deg,	P =   0.000 deg,	R =   90.000 deg
};
P[1575]{
   GP1:
	UF : 0, UT : 6,		CONFIG : 'N U T, 0, 0, 0',
	X =  249.606  mm,	Y =   -217.534  mm,	Z =   -258.361  mm,
	W =  90.000 deg,	P =   0.000 deg,	R =   90.000 deg
};
P[1576]{
   GP1:
	UF : 0, UT : 6,		CONFIG : 'N U T, 0, 0, 0',
	X =  248.622  mm,	Y =   -217.994  mm,	Z =   -258.180  mm,
	W =  90.000 deg,	P =   0.000 deg,	R =   90.000 deg
};
P[1577]{
   GP1:
	UF : 0, UT : 6,		CONFIG : 'N U T, 0, 0, 0',
	X =  247.625  mm,	Y =   -218.603  mm,	Z =   -258.377  mm,
	W =  90.000 deg,	P =   0.000 deg,	R =   90.000 deg
};
P[1578]{
   GP1:
	UF : 0, UT : 6,		CONFIG : 'N U T, 0, 0, 0',
	X =  246.729  mm,	Y =   -219.098  mm,	Z =   -258.247  mm,
	W =  90.000 deg,	P =   0.000 deg,	R =   90.000 deg
};
P[1579]{
   GP1:
	UF : 0, UT : 6,		CONFIG : 'N U T, 0, 0, 0',
	X =  245.672  mm,	Y =   -219.666  mm,	Z =   -257.986  mm,
	W =  90.000 deg,	P =   0.000 deg,	R =   90.000 deg
};
P[1580]{
   GP1:
	UF : 0, UT : 6,		CONFIG : 'N U T, 0, 0, 0',
	X =  245.205  mm,	Y =   -219.998  mm,	Z =   -258.364  mm,
	W =  90.000 deg,	P =   0.000 deg,	R =   90.000 deg
};
P[1581]{
   GP1:
	UF : 0, UT : 6,		CONFIG : 'N U T, 0, 0, 0',
	X =  244.427  mm,	Y =   -220.401  mm,	Z =   -258.078  mm,
	W =  90.000 deg,	P =   0.000 deg,	R =   90.000 deg
};
P[1582]{
   GP1:
	UF : 0, UT : 6,		CONFIG : 'N U T, 0, 0, 0',
	X =  243.930  mm,	Y =   -220.727  mm,	Z =   -258.323  mm,
	W =  90.000 deg,	P =   0.000 deg,	R =   90.000 deg
};
P[1583]{
   GP1:
	UF : 0, UT : 6,		CONFIG : 'N U T, 0, 0, 0',
	X =  242.903  mm,	Y =   -221.292  mm,	Z =   -258.150  mm,
	W =  90.000 deg,	P =   0.000 deg,	R =   90.000 deg
};
P[1584]{
   GP1:
	UF : 0, UT : 6,		CONFIG : 'N U T, 0, 0, 0',
	X =  241.926  mm,	Y =   -221.826  mm,	Z =   -257.962  mm,
	W =  90.000 deg,	P =   0.000 deg,	R =   90.000 deg
};
P[1585]{
   GP1:
	UF : 0, UT : 6,		CONFIG : 'N U T, 0, 0, 0',
	X =  241.339  mm,	Y =   -222.157  mm,	Z =   -257.914  mm,
	W =  90.000 deg,	P =   0.000 deg,	R =   90.000 deg
};
P[1586]{
   GP1:
	UF : 0, UT : 6,		CONFIG : 'N U T, 0, 0, 0',
	X =  239.518  mm,	Y =   -223.278  mm,	Z =   -258.345  mm,
	W =  90.000 deg,	P =   0.000 deg,	R =   90.000 deg
};
P[1587]{
   GP1:
	UF : 0, UT : 6,		CONFIG : 'N U T, 0, 0, 0',
	X =  236.453  mm,	Y =   -225.026  mm,	Z =   -258.215  mm,
	W =  90.000 deg,	P =   0.000 deg,	R =   90.000 deg
};
P[1588]{
   GP1:
	UF : 0, UT : 6,		CONFIG : 'N U T, 0, 0, 0',
	X =  235.618  mm,	Y =   -225.508  mm,	Z =   -258.205  mm,
	W =  90.000 deg,	P =   0.000 deg,	R =   90.000 deg
};
P[1589]{
   GP1:
	UF : 0, UT : 6,		CONFIG : 'N U T, 0, 0, 0',
	X =  232.427  mm,	Y =   -227.342  mm,	Z =   -258.159  mm,
	W =  90.000 deg,	P =   0.000 deg,	R =   90.000 deg
};
P[1590]{
   GP1:
	UF : 0, UT : 6,		CONFIG : 'N U T, 0, 0, 0',
	X =  231.680  mm,	Y =   -227.771  mm,	Z =   -258.144  mm,
	W =  90.000 deg,	P =   0.000 deg,	R =   90.000 deg
};
P[1591]{
   GP1:
	UF : 0, UT : 6,		CONFIG : 'N U T, 0, 0, 0',
	X =  230.607  mm,	Y =   -228.398  mm,	Z =   -258.195  mm,
	W =  90.000 deg,	P =   0.000 deg,	R =   90.000 deg
};
P[1592]{
   GP1:
	UF : 0, UT : 6,		CONFIG : 'N U T, 0, 0, 0',
	X =  229.725  mm,	Y =   -228.938  mm,	Z =   -258.377  mm,
	W =  90.000 deg,	P =   0.000 deg,	R =   90.000 deg
};
P[1593]{
   GP1:
	UF : 0, UT : 6,		CONFIG : 'N U T, 0, 0, 0',
	X =  226.150  mm,	Y =   -230.982  mm,	Z =   -258.252  mm,
	W =  90.000 deg,	P =   0.000 deg,	R =   90.000 deg
};
P[1594]{
   GP1:
	UF : 0, UT : 6,		CONFIG : 'N U T, 0, 0, 0',
	X =  224.985  mm,	Y =   -231.623  mm,	Z =   -258.058  mm,
	W =  90.000 deg,	P =   0.000 deg,	R =   90.000 deg
};
P[1595]{
   GP1:
	UF : 0, UT : 6,		CONFIG : 'N U T, 0, 0, 0',
	X =  224.403  mm,	Y =   -231.969  mm,	Z =   -258.123  mm,
	W =  90.000 deg,	P =   0.000 deg,	R =   90.000 deg
};
P[1596]{
   GP1:
	UF : 0, UT : 6,		CONFIG : 'N U T, 0, 0, 0',
	X =  223.636  mm,	Y =   -232.452  mm,	Z =   -258.366  mm,
	W =  90.000 deg,	P =   0.000 deg,	R =   90.000 deg
};
P[1597]{
   GP1:
	UF : 0, UT : 6,		CONFIG : 'N U T, 0, 0, 0',
	X =  221.933  mm,	Y =   -233.430  mm,	Z =   -258.340  mm,
	W =  90.000 deg,	P =   0.000 deg,	R =   90.000 deg
};
P[1598]{
   GP1:
	UF : 0, UT : 6,		CONFIG : 'N U T, 0, 0, 0',
	X =  220.901  mm,	Y =   -233.969  mm,	Z =   -257.989  mm,
	W =  90.000 deg,	P =   0.000 deg,	R =   90.000 deg
};
P[1599]{
   GP1:
	UF : 0, UT : 6,		CONFIG : 'N U T, 0, 0, 0',
	X =  219.621  mm,	Y =   -234.738  mm,	Z =   -258.171  mm,
	W =  90.000 deg,	P =   0.000 deg,	R =   90.000 deg
};
P[1600]{
   GP1:
	UF : 0, UT : 6,		CONFIG : 'N U T, 0, 0, 0',
	X =  218.082  mm,	Y =   -235.638  mm,	Z =   -258.238  mm,
	W =  90.000 deg,	P =   0.000 deg,	R =   90.000 deg
};
P[1601]{
   GP1:
	UF : 0, UT : 6,		CONFIG : 'N U T, 0, 0, 0',
	X =  215.684  mm,	Y =   -237.036  mm,	Z =   -258.325  mm,
	W =  90.000 deg,	P =   0.000 deg,	R =   90.000 deg
};
P[1602]{
   GP1:
	UF : 0, UT : 6,		CONFIG : 'N U T, 0, 0, 0',
	X =  214.711  mm,	Y =   -237.551  mm,	Z =   -258.038  mm,
	W =  90.000 deg,	P =   0.000 deg,	R =   90.000 deg
};
P[1603]{
   GP1:
	UF : 0, UT : 6,		CONFIG : 'N U T, 0, 0, 0',
	X =  213.993  mm,	Y =   -237.945  mm,	Z =   -257.913  mm,
	W =  90.000 deg,	P =   0.000 deg,	R =   90.000 deg
};
P[1604]{
   GP1:
	UF : 0, UT : 6,		CONFIG : 'N U T, 0, 0, 0',
	X =  213.059  mm,	Y =   -238.559  mm,	Z =   -258.371  mm,
	W =  90.000 deg,	P =   0.000 deg,	R =   90.000 deg
};
P[1605]{
   GP1:
	UF : 0, UT : 6,		CONFIG : 'N U T, 0, 0, 0',
	X =  211.660  mm,	Y =   -239.355  mm,	Z =   -258.299  mm,
	W =  90.000 deg,	P =   0.000 deg,	R =   90.000 deg
};
P[1606]{
   GP1:
	UF : 0, UT : 6,		CONFIG : 'N U T, 0, 0, 0',
	X =  210.781  mm,	Y =   -239.825  mm,	Z =   -258.066  mm,
	W =  90.000 deg,	P =   0.000 deg,	R =   90.000 deg
};
P[1607]{
   GP1:
	UF : 0, UT : 6,		CONFIG : 'N U T, 0, 0, 0',
	X =  209.277  mm,	Y =   -240.673  mm,	Z =   -257.938  mm,
	W =  90.000 deg,	P =   0.000 deg,	R =   90.000 deg
};
P[1608]{
   GP1:
	UF : 0, UT : 6,		CONFIG : 'N U T, 0, 0, 0',
	X =  206.199  mm,	Y =   -242.463  mm,	Z =   -258.015  mm,
	W =  90.000 deg,	P =   0.000 deg,	R =   90.000 deg
};
P[1609]{
   GP1:
	UF : 0, UT : 6,		CONFIG : 'N U T, 0, 0, 0',
	X =  204.442  mm,	Y =   -243.459  mm,	Z =   -257.901  mm,
	W =  90.000 deg,	P =   0.000 deg,	R =   90.000 deg
};
P[1610]{
   GP1:
	UF : 0, UT : 6,		CONFIG : 'N U T, 0, 0, 0',
	X =  203.730  mm,	Y =   -243.947  mm,	Z =   -258.379  mm,
	W =  90.000 deg,	P =   0.000 deg,	R =   90.000 deg
};
P[1611]{
   GP1:
	UF : 0, UT : 6,		CONFIG : 'N U T, 0, 0, 0',
	X =  202.292  mm,	Y =   -244.770  mm,	Z =   -258.336  mm,
	W =  90.000 deg,	P =   0.000 deg,	R =   90.000 deg
};
P[1612]{
   GP1:
	UF : 0, UT : 6,		CONFIG : 'N U T, 0, 0, 0',
	X =  201.484  mm,	Y =   -245.225  mm,	Z =   -258.261  mm,
	W =  90.000 deg,	P =   0.000 deg,	R =   90.000 deg
};
P[1613]{
   GP1:
	UF : 0, UT : 6,		CONFIG : 'N U T, 0, 0, 0',
	X =  200.804  mm,	Y =   -245.584  mm,	Z =   -258.053  mm,
	W =  90.000 deg,	P =   0.000 deg,	R =   90.000 deg
};
P[1614]{
   GP1:
	UF : 0, UT : 6,		CONFIG : 'N U T, 0, 0, 0',
	X =  199.705  mm,	Y =   -246.260  mm,	Z =   -258.314  mm,
	W =  90.000 deg,	P =   0.000 deg,	R =   90.000 deg
};
P[1615]{
   GP1:
	UF : 0, UT : 6,		CONFIG : 'N U T, 0, 0, 0',
	X =  198.107  mm,	Y =   -247.157  mm,	Z =   -258.153  mm,
	W =  90.000 deg,	P =   0.000 deg,	R =   90.000 deg
};
P[1616]{
   GP1:
	UF : 0, UT : 6,		CONFIG : 'N U T, 0, 0, 0',
	X =  196.850  mm,	Y =   -247.843  mm,	Z =   -257.913  mm,
	W =  90.000 deg,	P =   0.000 deg,	R =   90.000 deg
};
P[1617]{
   GP1:
	UF : 0, UT : 6,		CONFIG : 'N U T, 0, 0, 0',
	X =  195.707  mm,	Y =   -248.504  mm,	Z =   -257.910  mm,
	W =  90.000 deg,	P =   0.000 deg,	R =   90.000 deg
};
P[1618]{
   GP1:
	UF : 0, UT : 6,		CONFIG : 'N U T, 0, 0, 0',
	X =  194.098  mm,	Y =   -249.463  mm,	Z =   -258.102  mm,
	W =  90.000 deg,	P =   0.000 deg,	R =   90.000 deg
};
P[1619]{
   GP1:
	UF : 0, UT : 6,		CONFIG : 'N U T, 0, 0, 0',
	X =  193.056  mm,	Y =   -250.042  mm,	Z =   -257.958  mm,
	W =  90.000 deg,	P =   0.000 deg,	R =   90.000 deg
};
P[1620]{
   GP1:
	UF : 0, UT : 6,		CONFIG : 'N U T, 0, 0, 0',
	X =  187.970  mm,	Y =   -252.993  mm,	Z =   -258.046  mm,
	W =  90.000 deg,	P =   0.000 deg,	R =   90.000 deg
};
P[1621]{
   GP1:
	UF : 0, UT : 6,		CONFIG : 'N U T, 0, 0, 0',
	X =  187.024  mm,	Y =   -253.532  mm,	Z =   -258.000  mm,
	W =  90.000 deg,	P =   0.000 deg,	R =   90.000 deg
};
P[1622]{
   GP1:
	UF : 0, UT : 6,		CONFIG : 'N U T, 0, 0, 0',
	X =  184.836  mm,	Y =   -254.805  mm,	Z =   -258.059  mm,
	W =  90.000 deg,	P =   0.000 deg,	R =   90.000 deg
};
P[1623]{
   GP1:
	UF : 0, UT : 6,		CONFIG : 'N U T, 0, 0, 0',
	X =  183.185  mm,	Y =   -255.790  mm,	Z =   -258.262  mm,
	W =  90.000 deg,	P =   0.000 deg,	R =   90.000 deg
};
P[1624]{
   GP1:
	UF : 0, UT : 6,		CONFIG : 'N U T, 0, 0, 0',
	X =  182.379  mm,	Y =   -256.270  mm,	Z =   -258.343  mm,
	W =  90.000 deg,	P =   0.000 deg,	R =   90.000 deg
};
P[1625]{
   GP1:
	UF : 0, UT : 6,		CONFIG : 'N U T, 0, 0, 0',
	X =  180.459  mm,	Y =   -257.331  mm,	Z =   -258.052  mm,
	W =  90.000 deg,	P =   0.000 deg,	R =   90.000 deg
};
P[1626]{
   GP1:
	UF : 0, UT : 6,		CONFIG : 'N U T, 0, 0, 0',
	X =  178.877  mm,	Y =   -258.245  mm,	Z =   -258.055  mm,
	W =  90.000 deg,	P =   0.000 deg,	R =   90.000 deg
};
P[1627]{
   GP1:
	UF : 0, UT : 6,		CONFIG : 'N U T, 0, 0, 0',
	X =  177.926  mm,	Y =   -258.838  mm,	Z =   -258.333  mm,
	W =  90.000 deg,	P =   0.000 deg,	R =   90.000 deg
};
P[1628]{
   GP1:
	UF : 0, UT : 6,		CONFIG : 'N U T, 0, 0, 0',
	X =  175.867  mm,	Y =   -260.033  mm,	Z =   -258.361  mm,
	W =  90.000 deg,	P =   0.000 deg,	R =   90.000 deg
};
P[1629]{
   GP1:
	UF : 0, UT : 6,		CONFIG : 'N U T, 0, 0, 0',
	X =  174.921  mm,	Y =   -260.522  mm,	Z =   -258.012  mm,
	W =  90.000 deg,	P =   0.000 deg,	R =   90.000 deg
};
P[1630]{
   GP1:
	UF : 0, UT : 6,		CONFIG : 'N U T, 0, 0, 0',
	X =  173.678  mm,	Y =   -261.240  mm,	Z =   -258.019  mm,
	W =  90.000 deg,	P =   0.000 deg,	R =   90.000 deg
};
P[1631]{
   GP1:
	UF : 0, UT : 6,		CONFIG : 'N U T, 0, 0, 0',
	X =  172.378  mm,	Y =   -262.029  mm,	Z =   -258.249  mm,
	W =  90.000 deg,	P =   0.000 deg,	R =   90.000 deg
};
P[1632]{
   GP1:
	UF : 0, UT : 6,		CONFIG : 'N U T, 0, 0, 0',
	X =  170.903  mm,	Y =   -262.858  mm,	Z =   -258.111  mm,
	W =  90.000 deg,	P =   0.000 deg,	R =   90.000 deg
};
P[1633]{
   GP1:
	UF : 0, UT : 6,		CONFIG : 'N U T, 0, 0, 0',
	X =  169.963  mm,	Y =   -263.393  mm,	Z =   -258.064  mm,
	W =  90.000 deg,	P =   0.000 deg,	R =   90.000 deg
};
P[1634]{
   GP1:
	UF : 0, UT : 6,		CONFIG : 'N U T, 0, 0, 0',
	X =  169.293  mm,	Y =   -263.822  mm,	Z =   -258.323  mm,
	W =  90.000 deg,	P =   0.000 deg,	R =   90.000 deg
};
P[1635]{
   GP1:
	UF : 0, UT : 6,		CONFIG : 'N U T, 0, 0, 0',
	X =  168.266  mm,	Y =   -264.389  mm,	Z =   -258.167  mm,
	W =  90.000 deg,	P =   0.000 deg,	R =   90.000 deg
};
P[1636]{
   GP1:
	UF : 0, UT : 6,		CONFIG : 'N U T, 0, 0, 0',
	X =  165.161  mm,	Y =   -266.216  mm,	Z =   -258.376  mm,
	W =  90.000 deg,	P =   0.000 deg,	R =   90.000 deg
};
P[1637]{
   GP1:
	UF : 0, UT : 6,		CONFIG : 'N U T, 0, 0, 0',
	X =  164.648  mm,	Y =   -266.448  mm,	Z =   -257.977  mm,
	W =  90.000 deg,	P =   0.000 deg,	R =   90.000 deg
};
P[1638]{
   GP1:
	UF : 0, UT : 6,		CONFIG : 'N U T, 0, 0, 0',
	X =  159.613  mm,	Y =   -269.404  mm,	Z =   -258.279  mm,
	W =  90.000 deg,	P =   0.000 deg,	R =   90.000 deg
};
P[1639]{
   GP1:
	UF : 0, UT : 6,		CONFIG : 'N U T, 0, 0, 0',
	X =  158.097  mm,	Y =   -270.263  mm,	Z =   -258.177  mm,
	W =  90.000 deg,	P =   0.000 deg,	R =   90.000 deg
};
P[1640]{
   GP1:
	UF : 0, UT : 6,		CONFIG : 'N U T, 0, 0, 0',
	X =  156.323  mm,	Y =   -271.298  mm,	Z =   -258.248  mm,
	W =  90.000 deg,	P =   0.000 deg,	R =   90.000 deg
};
P[1641]{
   GP1:
	UF : 0, UT : 6,		CONFIG : 'N U T, 0, 0, 0',
	X =  155.685  mm,	Y =   -271.672  mm,	Z =   -258.282  mm,
	W =  90.000 deg,	P =   0.000 deg,	R =   90.000 deg
};
P[1642]{
   GP1:
	UF : 0, UT : 6,		CONFIG : 'N U T, 0, 0, 0',
	X =  152.411  mm,	Y =   -273.503  mm,	Z =   -257.918  mm,
	W =  90.000 deg,	P =   0.000 deg,	R =   90.000 deg
};
P[1643]{
   GP1:
	UF : 0, UT : 6,		CONFIG : 'N U T, 0, 0, 0',
	X =  151.686  mm,	Y =   -273.974  mm,	Z =   -258.235  mm,
	W =  90.000 deg,	P =   0.000 deg,	R =   90.000 deg
};
P[1644]{
   GP1:
	UF : 0, UT : 6,		CONFIG : 'N U T, 0, 0, 0',
	X =  148.949  mm,	Y =   -274.676  mm,	Z =   -252.823  mm,
	W =  90.000 deg,	P =   0.000 deg,	R =   90.000 deg
};
P[1645]{
   GP1:
	UF : 0, UT : 6,		CONFIG : 'N U T, 0, 0, 0',
	X =  148.154  mm,	Y =   -275.095  mm,	Z =   -252.574  mm,
	W =  90.000 deg,	P =   0.000 deg,	R =   90.000 deg
};
P[1646]{
   GP1:
	UF : 0, UT : 6,		CONFIG : 'N U T, 0, 0, 0',
	X =  147.434  mm,	Y =   -275.513  mm,	Z =   -252.592  mm,
	W =  90.000 deg,	P =   0.000 deg,	R =   90.000 deg
};
P[1647]{
   GP1:
	UF : 0, UT : 6,		CONFIG : 'N U T, 0, 0, 0',
	X =  143.214  mm,	Y =   -277.985  mm,	Z =   -252.809  mm,
	W =  90.000 deg,	P =   0.000 deg,	R =   90.000 deg
};
P[1648]{
   GP1:
	UF : 0, UT : 6,		CONFIG : 'N U T, 0, 0, 0',
	X =  141.549  mm,	Y =   -278.933  mm,	Z =   -252.726  mm,
	W =  90.000 deg,	P =   0.000 deg,	R =   90.000 deg
};
P[1649]{
   GP1:
	UF : 0, UT : 6,		CONFIG : 'N U T, 0, 0, 0',
	X =  140.800  mm,	Y =   -279.309  mm,	Z =   -252.375  mm,
	W =  90.000 deg,	P =   0.000 deg,	R =   90.000 deg
};
P[1650]{
   GP1:
	UF : 0, UT : 6,		CONFIG : 'N U T, 0, 0, 0',
	X =  138.526  mm,	Y =   -280.691  mm,	Z =   -252.805  mm,
	W =  90.000 deg,	P =   0.000 deg,	R =   90.000 deg
};
P[1651]{
   GP1:
	UF : 0, UT : 6,		CONFIG : 'N U T, 0, 0, 0',
	X =  137.678  mm,	Y =   -281.171  mm,	Z =   -252.744  mm,
	W =  90.000 deg,	P =   0.000 deg,	R =   90.000 deg
};
P[1652]{
   GP1:
	UF : 0, UT : 6,		CONFIG : 'N U T, 0, 0, 0',
	X =  136.146  mm,	Y =   -282.031  mm,	Z =   -252.595  mm,
	W =  90.000 deg,	P =   0.000 deg,	R =   90.000 deg
};
P[1653]{
   GP1:
	UF : 0, UT : 6,		CONFIG : 'N U T, 0, 0, 0',
	X =  135.119  mm,	Y =   -282.598  mm,	Z =   -252.430  mm,
	W =  90.000 deg,	P =   0.000 deg,	R =   90.000 deg
};
P[1654]{
   GP1:
	UF : 0, UT : 6,		CONFIG : 'N U T, 0, 0, 0',
	X =  134.253  mm,	Y =   -283.158  mm,	Z =   -252.803  mm,
	W =  90.000 deg,	P =   0.000 deg,	R =   90.000 deg
};
P[1655]{
   GP1:
	UF : 0, UT : 6,		CONFIG : 'N U T, 0, 0, 0',
	X =  133.309  mm,	Y =   -283.644  mm,	Z =   -252.436  mm,
	W =  90.000 deg,	P =   0.000 deg,	R =   90.000 deg
};
P[1656]{
   GP1:
	UF : 0, UT : 6,		CONFIG : 'N U T, 0, 0, 0',
	X =  132.119  mm,	Y =   -284.390  mm,	Z =   -252.807  mm,
	W =  90.000 deg,	P =   0.000 deg,	R =   90.000 deg
};
P[1657]{
   GP1:
	UF : 0, UT : 6,		CONFIG : 'N U T, 0, 0, 0',
	X =  129.714  mm,	Y =   -285.760  mm,	Z =   -252.690  mm,
	W =  90.000 deg,	P =   0.000 deg,	R =   90.000 deg
};
P[1658]{
   GP1:
	UF : 0, UT : 6,		CONFIG : 'N U T, 0, 0, 0',
	X =  128.788  mm,	Y =   -286.304  mm,	Z =   -252.748  mm,
	W =  90.000 deg,	P =   0.000 deg,	R =   90.000 deg
};
P[1659]{
   GP1:
	UF : 0, UT : 6,		CONFIG : 'N U T, 0, 0, 0',
	X =  127.263  mm,	Y =   -287.134  mm,	Z =   -252.436  mm,
	W =  90.000 deg,	P =   0.000 deg,	R =   90.000 deg
};
P[1660]{
   GP1:
	UF : 0, UT : 6,		CONFIG : 'N U T, 0, 0, 0',
	X =  126.466  mm,	Y =   -287.621  mm,	Z =   -252.598  mm,
	W =  90.000 deg,	P =   0.000 deg,	R =   90.000 deg
};
P[1661]{
   GP1:
	UF : 0, UT : 6,		CONFIG : 'N U T, 0, 0, 0',
	X =  125.395  mm,	Y =   -288.230  mm,	Z =   -252.544  mm,
	W =  90.000 deg,	P =   0.000 deg,	R =   90.000 deg
};
P[1662]{
   GP1:
	UF : 0, UT : 6,		CONFIG : 'N U T, 0, 0, 0',
	X =  123.382  mm,	Y =   -289.429  mm,	Z =   -252.769  mm,
	W =  90.000 deg,	P =   0.000 deg,	R =   90.000 deg
};
P[1663]{
   GP1:
	UF : 0, UT : 6,		CONFIG : 'N U T, 0, 0, 0',
	X =  122.513  mm,	Y =   -289.906  mm,	Z =   -252.615  mm,
	W =  90.000 deg,	P =   0.000 deg,	R =   90.000 deg
};
P[1664]{
   GP1:
	UF : 0, UT : 6,		CONFIG : 'N U T, 0, 0, 0',
	X =  118.561  mm,	Y =   -292.169  mm,	Z =   -252.501  mm,
	W =  90.000 deg,	P =   0.000 deg,	R =   90.000 deg
};
P[1665]{
   GP1:
	UF : 0, UT : 6,		CONFIG : 'N U T, 0, 0, 0',
	X =  117.569  mm,	Y =   -292.755  mm,	Z =   -252.580  mm,
	W =  90.000 deg,	P =   0.000 deg,	R =   90.000 deg
};
P[1666]{
   GP1:
	UF : 0, UT : 6,		CONFIG : 'N U T, 0, 0, 0',
	X =  116.135  mm,	Y =   -293.604  mm,	Z =   -252.711  mm,
	W =  90.000 deg,	P =   0.000 deg,	R =   90.000 deg
};
P[1667]{
   GP1:
	UF : 0, UT : 6,		CONFIG : 'N U T, 0, 0, 0',
	X =  114.438  mm,	Y =   -294.594  mm,	Z =   -252.776  mm,
	W =  90.000 deg,	P =   0.000 deg,	R =   90.000 deg
};
P[1668]{
   GP1:
	UF : 0, UT : 6,		CONFIG : 'N U T, 0, 0, 0',
	X =  107.948  mm,	Y =   -298.320  mm,	Z =   -252.641  mm,
	W =  90.000 deg,	P =   0.000 deg,	R =   90.000 deg
};
P[1669]{
   GP1:
	UF : 0, UT : 6,		CONFIG : 'N U T, 0, 0, 0',
	X =  104.937  mm,	Y =   -300.085  mm,	Z =   -252.805  mm,
	W =  90.000 deg,	P =   0.000 deg,	R =   90.000 deg
};
P[1670]{
   GP1:
	UF : 0, UT : 6,		CONFIG : 'N U T, 0, 0, 0',
	X =  102.458  mm,	Y =   -301.493  mm,	Z =   -252.659  mm,
	W =  90.000 deg,	P =   0.000 deg,	R =   90.000 deg
};
P[1671]{
   GP1:
	UF : 0, UT : 6,		CONFIG : 'N U T, 0, 0, 0',
	X =  101.522  mm,	Y =   -302.031  mm,	Z =   -252.651  mm,
	W =  90.000 deg,	P =   0.000 deg,	R =   90.000 deg
};
P[1672]{
   GP1:
	UF : 0, UT : 6,		CONFIG : 'N U T, 0, 0, 0',
	X =  99.921  mm,	Y =   -302.978  mm,	Z =   -252.788  mm,
	W =  90.000 deg,	P =   0.000 deg,	R =   90.000 deg
};
P[1673]{
   GP1:
	UF : 0, UT : 6,		CONFIG : 'N U T, 0, 0, 0',
	X =  99.325  mm,	Y =   -303.290  mm,	Z =   -252.591  mm,
	W =  90.000 deg,	P =   0.000 deg,	R =   90.000 deg
};
P[1674]{
   GP1:
	UF : 0, UT : 6,		CONFIG : 'N U T, 0, 0, 0',
	X =  98.587  mm,	Y =   -303.738  mm,	Z =   -252.729  mm,
	W =  90.000 deg,	P =   0.000 deg,	R =   90.000 deg
};
P[1675]{
   GP1:
	UF : 0, UT : 6,		CONFIG : 'N U T, 0, 0, 0',
	X =  97.707  mm,	Y =   -304.258  mm,	Z =   -252.797  mm,
	W =  90.000 deg,	P =   0.000 deg,	R =   90.000 deg
};
P[1676]{
   GP1:
	UF : 0, UT : 6,		CONFIG : 'N U T, 0, 0, 0',
	X =  96.061  mm,	Y =   -305.156  mm,	Z =   -252.479  mm,
	W =  90.000 deg,	P =   0.000 deg,	R =   90.000 deg
};
P[1677]{
   GP1:
	UF : 0, UT : 6,		CONFIG : 'N U T, 0, 0, 0',
	X =  93.582  mm,	Y =   -306.636  mm,	Z =   -252.775  mm,
	W =  90.000 deg,	P =   0.000 deg,	R =   90.000 deg
};
P[1678]{
   GP1:
	UF : 0, UT : 6,		CONFIG : 'N U T, 0, 0, 0',
	X =  92.203  mm,	Y =   -307.405  mm,	Z =   -252.606  mm,
	W =  90.000 deg,	P =   0.000 deg,	R =   90.000 deg
};
P[1679]{
   GP1:
	UF : 0, UT : 6,		CONFIG : 'N U T, 0, 0, 0',
	X =  91.541  mm,	Y =   -307.798  mm,	Z =   -252.674  mm,
	W =  90.000 deg,	P =   0.000 deg,	R =   90.000 deg
};
P[1680]{
   GP1:
	UF : 0, UT : 6,		CONFIG : 'N U T, 0, 0, 0',
	X =  89.738  mm,	Y =   -308.831  mm,	Z =   -252.622  mm,
	W =  90.000 deg,	P =   0.000 deg,	R =   90.000 deg
};
P[1681]{
   GP1:
	UF : 0, UT : 6,		CONFIG : 'N U T, 0, 0, 0',
	X =  86.377  mm,	Y =   -310.738  mm,	Z =   -252.408  mm,
	W =  90.000 deg,	P =   0.000 deg,	R =   90.000 deg
};
P[1682]{
   GP1:
	UF : 0, UT : 6,		CONFIG : 'N U T, 0, 0, 0',
	X =  85.588  mm,	Y =   -311.189  mm,	Z =   -252.394  mm,
	W =  90.000 deg,	P =   0.000 deg,	R =   90.000 deg
};
P[1683]{
   GP1:
	UF : 0, UT : 6,		CONFIG : 'N U T, 0, 0, 0',
	X =  84.710  mm,	Y =   -311.716  mm,	Z =   -252.510  mm,
	W =  90.000 deg,	P =   0.000 deg,	R =   90.000 deg
};
P[1684]{
   GP1:
	UF : 0, UT : 6,		CONFIG : 'N U T, 0, 0, 0',
	X =  83.575  mm,	Y =   -312.420  mm,	Z =   -252.807  mm,
	W =  90.000 deg,	P =   0.000 deg,	R =   90.000 deg
};
P[1685]{
   GP1:
	UF : 0, UT : 6,		CONFIG : 'N U T, 0, 0, 0',
	X =  81.983  mm,	Y =   -313.302  mm,	Z =   -252.580  mm,
	W =  90.000 deg,	P =   0.000 deg,	R =   90.000 deg
};
P[1686]{
   GP1:
	UF : 0, UT : 6,		CONFIG : 'N U T, 0, 0, 0',
	X =  80.646  mm,	Y =   -314.055  mm,	Z =   -252.462  mm,
	W =  90.000 deg,	P =   0.000 deg,	R =   90.000 deg
};
P[1687]{
   GP1:
	UF : 0, UT : 6,		CONFIG : 'N U T, 0, 0, 0',
	X =  78.463  mm,	Y =   -315.322  mm,	Z =   -252.506  mm,
	W =  90.000 deg,	P =   0.000 deg,	R =   90.000 deg
};
P[1688]{
   GP1:
	UF : 0, UT : 6,		CONFIG : 'N U T, 0, 0, 0',
	X =  77.522  mm,	Y =   -315.883  mm,	Z =   -252.616  mm,
	W =  90.000 deg,	P =   0.000 deg,	R =   90.000 deg
};
P[1689]{
   GP1:
	UF : 0, UT : 6,		CONFIG : 'N U T, 0, 0, 0',
	X =  75.522  mm,	Y =   -317.027  mm,	Z =   -252.549  mm,
	W =  90.000 deg,	P =   0.000 deg,	R =   90.000 deg
};
P[1690]{
   GP1:
	UF : 0, UT : 6,		CONFIG : 'N U T, 0, 0, 0',
	X =  74.896  mm,	Y =   -317.392  mm,	Z =   -252.565  mm,
	W =  90.000 deg,	P =   0.000 deg,	R =   90.000 deg
};
P[1691]{
   GP1:
	UF : 0, UT : 6,		CONFIG : 'N U T, 0, 0, 0',
	X =  73.985  mm,	Y =   -317.944  mm,	Z =   -252.726  mm,
	W =  90.000 deg,	P =   0.000 deg,	R =   90.000 deg
};
P[1692]{
   GP1:
	UF : 0, UT : 6,		CONFIG : 'N U T, 0, 0, 0',
	X =  73.010  mm,	Y =   -318.512  mm,	Z =   -252.756  mm,
	W =  90.000 deg,	P =   0.000 deg,	R =   90.000 deg
};
P[1693]{
   GP1:
	UF : 0, UT : 6,		CONFIG : 'N U T, 0, 0, 0',
	X =  71.585  mm,	Y =   -319.339  mm,	Z =   -252.784  mm,
	W =  90.000 deg,	P =   0.000 deg,	R =   90.000 deg
};
P[1694]{
   GP1:
	UF : 0, UT : 6,		CONFIG : 'N U T, 0, 0, 0',
	X =  70.436  mm,	Y =   -319.973  mm,	Z =   -252.610  mm,
	W =  90.000 deg,	P =   0.000 deg,	R =   90.000 deg
};
P[1695]{
   GP1:
	UF : 0, UT : 6,		CONFIG : 'N U T, 0, 0, 0',
	X =  69.687  mm,	Y =   -320.420  mm,	Z =   -252.691  mm,
	W =  90.000 deg,	P =   0.000 deg,	R =   90.000 deg
};
P[1696]{
   GP1:
	UF : 0, UT : 6,		CONFIG : 'N U T, 0, 0, 0',
	X =  68.040  mm,	Y =   -321.388  mm,	Z =   -252.802  mm,
	W =  90.000 deg,	P =   0.000 deg,	R =   90.000 deg
};
P[1697]{
   GP1:
	UF : 0, UT : 6,		CONFIG : 'N U T, 0, 0, 0',
	X =  67.446  mm,	Y =   -321.694  mm,	Z =   -252.570  mm,
	W =  90.000 deg,	P =   0.000 deg,	R =   90.000 deg
};
P[1698]{
   GP1:
	UF : 0, UT : 6,		CONFIG : 'N U T, 0, 0, 0',
	X =  66.497  mm,	Y =   -322.219  mm,	Z =   -252.432  mm,
	W =  90.000 deg,	P =   0.000 deg,	R =   90.000 deg
};
P[1699]{
   GP1:
	UF : 0, UT : 6,		CONFIG : 'N U T, 0, 0, 0',
	X =  65.885  mm,	Y =   -322.600  mm,	Z =   -252.599  mm,
	W =  90.000 deg,	P =   0.000 deg,	R =   90.000 deg
};
P[1700]{
   GP1:
	UF : 0, UT : 6,		CONFIG : 'N U T, 0, 0, 0',
	X =  64.997  mm,	Y =   -323.122  mm,	Z =   -252.660  mm,
	W =  90.000 deg,	P =   0.000 deg,	R =   90.000 deg
};
P[1701]{
   GP1:
	UF : 0, UT : 6,		CONFIG : 'N U T, 0, 0, 0',
	X =  63.613  mm,	Y =   -323.883  mm,	Z =   -252.425  mm,
	W =  90.000 deg,	P =   0.000 deg,	R =   90.000 deg
};
P[1702]{
   GP1:
	UF : 0, UT : 6,		CONFIG : 'N U T, 0, 0, 0',
	X =  62.059  mm,	Y =   -324.789  mm,	Z =   -252.477  mm,
	W =  90.000 deg,	P =   0.000 deg,	R =   90.000 deg
};
P[1703]{
   GP1:
	UF : 0, UT : 6,		CONFIG : 'N U T, 0, 0, 0',
	X =  59.357  mm,	Y =   -326.406  mm,	Z =   -252.830  mm,
	W =  90.000 deg,	P =   0.000 deg,	R =   90.000 deg
};
P[1704]{
   GP1:
	UF : 0, UT : 6,		CONFIG : 'N U T, 0, 0, 0',
	X =  57.532  mm,	Y =   -327.390  mm,	Z =   -252.398  mm,
	W =  90.000 deg,	P =   0.000 deg,	R =   90.000 deg
};
P[1705]{
   GP1:
	UF : 0, UT : 6,		CONFIG : 'N U T, 0, 0, 0',
	X =  56.057  mm,	Y =   -328.233  mm,	Z =   -252.344  mm,
	W =  90.000 deg,	P =   0.000 deg,	R =   90.000 deg
};
P[1706]{
   GP1:
	UF : 0, UT : 6,		CONFIG : 'N U T, 0, 0, 0',
	X =  55.021  mm,	Y =   -328.906  mm,	Z =   -252.802  mm,
	W =  90.000 deg,	P =   0.000 deg,	R =   90.000 deg
};
P[1707]{
   GP1:
	UF : 0, UT : 6,		CONFIG : 'N U T, 0, 0, 0',
	X =  54.277  mm,	Y =   -329.318  mm,	Z =   -252.699  mm,
	W =  90.000 deg,	P =   0.000 deg,	R =   90.000 deg
};
P[1708]{
   GP1:
	UF : 0, UT : 6,		CONFIG : 'N U T, 0, 0, 0',
	X =  51.727  mm,	Y =   -329.729  mm,	Z =   -252.631  mm,
	W =  90.000 deg,	P =   0.000 deg,	R =   90.000 deg
};
P[1709]{
   GP1:
	UF : 0, UT : 6,		CONFIG : 'N U T, 0, 0, 0',
	X =  52.276  mm,	Y =   -330.601  mm,	Z =   -252.506  mm,
	W =  90.000 deg,	P =   0.000 deg,	R =   90.000 deg
};
P[1710]{
   GP1:
	UF : 0, UT : 6,		CONFIG : 'N U T, 0, 0, 0',
	X =  50.574  mm,	Y =   -330.838  mm,	Z =   -252.611  mm,
	W =  90.000 deg,	P =   0.000 deg,	R =   90.000 deg
};
P[1711]{
   GP1:
	UF : 0, UT : 6,		CONFIG : 'N U T, 0, 0, 0',
	X =  51.823  mm,	Y =   -331.198  mm,	Z =   -252.563  mm,
	W =  90.000 deg,	P =   0.000 deg,	R =   90.000 deg
};
P[1712]{
   GP1:
	UF : 0, UT : 6,		CONFIG : 'N U T, 0, 0, 0',
	X =  51.422  mm,	Y =   -331.916  mm,	Z =   -252.528  mm,
	W =  90.000 deg,	P =   0.000 deg,	R =   90.000 deg
};
P[1713]{
   GP1:
	UF : 0, UT : 6,		CONFIG : 'N U T, 0, 0, 0',
	X =  50.106  mm,	Y =   -331.745  mm,	Z =   -252.663  mm,
	W =  90.000 deg,	P =   0.000 deg,	R =   90.000 deg
};
P[1714]{
   GP1:
	UF : 0, UT : 6,		CONFIG : 'N U T, 0, 0, 0',
	X =  51.226  mm,	Y =   -332.571  mm,	Z =   -252.744  mm,
	W =  90.000 deg,	P =   0.000 deg,	R =   90.000 deg
};
P[1715]{
   GP1:
	UF : 0, UT : 6,		CONFIG : 'N U T, 0, 0, 0',
	X =  49.832  mm,	Y =   -333.094  mm,	Z =   -252.706  mm,
	W =  90.000 deg,	P =   0.000 deg,	R =   90.000 deg
};
P[1716]{
   GP1:
	UF : 0, UT : 6,		CONFIG : 'N U T, 0, 0, 0',
	X =  49.941  mm,	Y =   -334.041  mm,	Z =   -252.744  mm,
	W =  90.000 deg,	P =   0.000 deg,	R =   90.000 deg
};
P[1717]{
   GP1:
	UF : 0, UT : 6,		CONFIG : 'N U T, 0, 0, 0',
	X =  50.319  mm,	Y =   -335.071  mm,	Z =   -252.798  mm,
	W =  90.000 deg,	P =   0.000 deg,	R =   90.000 deg
};
P[1718]{
   GP1:
	UF : 0, UT : 6,		CONFIG : 'N U T, 0, 0, 0',
	X =  51.613  mm,	Y =   -335.422  mm,	Z =   -252.833  mm,
	W =  90.000 deg,	P =   0.000 deg,	R =   90.000 deg
};
P[1719]{
   GP1:
	UF : 0, UT : 6,		CONFIG : 'N U T, 0, 0, 0',
	X =  52.078  mm,	Y =   -336.409  mm,	Z =   -252.421  mm,
	W =  90.000 deg,	P =   0.000 deg,	R =   90.000 deg
};
P[1720]{
   GP1:
	UF : 0, UT : 6,		CONFIG : 'N U T, 0, 0, 0',
	X =  52.522  mm,	Y =   -337.121  mm,	Z =   -252.624  mm,
	W =  90.000 deg,	P =   0.000 deg,	R =   90.000 deg
};
P[1721]{
   GP1:
	UF : 0, UT : 6,		CONFIG : 'N U T, 0, 0, 0',
	X =  53.957  mm,	Y =   -339.561  mm,	Z =   -252.781  mm,
	W =  90.000 deg,	P =   0.000 deg,	R =   90.000 deg
};
P[1722]{
   GP1:
	UF : 0, UT : 6,		CONFIG : 'N U T, 0, 0, 0',
	X =  54.518  mm,	Y =   -340.606  mm,	Z =   -252.525  mm,
	W =  90.000 deg,	P =   0.000 deg,	R =   90.000 deg
};
P[1723]{
   GP1:
	UF : 0, UT : 6,		CONFIG : 'N U T, 0, 0, 0',
	X =  54.872  mm,	Y =   -341.250  mm,	Z =   -252.418  mm,
	W =  90.000 deg,	P =   0.000 deg,	R =   90.000 deg
};
P[1724]{
   GP1:
	UF : 0, UT : 6,		CONFIG : 'N U T, 0, 0, 0',
	X =  55.349  mm,	Y =   -342.055  mm,	Z =   -252.489  mm,
	W =  90.000 deg,	P =   0.000 deg,	R =   90.000 deg
};
P[1725]{
   GP1:
	UF : 0, UT : 6,		CONFIG : 'N U T, 0, 0, 0',
	X =  56.042  mm,	Y =   -343.246  mm,	Z =   -252.525  mm,
	W =  90.000 deg,	P =   0.000 deg,	R =   90.000 deg
};
P[1726]{
   GP1:
	UF : 0, UT : 6,		CONFIG : 'N U T, 0, 0, 0',
	X =  56.648  mm,	Y =   -344.256  mm,	Z =   -252.670  mm,
	W =  90.000 deg,	P =   0.000 deg,	R =   90.000 deg
};
P[1727]{
   GP1:
	UF : 0, UT : 6,		CONFIG : 'N U T, 0, 0, 0',
	X =  57.551  mm,	Y =   -345.813  mm,	Z =   -252.690  mm,
	W =  90.000 deg,	P =   0.000 deg,	R =   90.000 deg
};
P[1728]{
   GP1:
	UF : 0, UT : 6,		CONFIG : 'N U T, 0, 0, 0',
	X =  58.380  mm,	Y =   -347.341  mm,	Z =   -252.360  mm,
	W =  90.000 deg,	P =   0.000 deg,	R =   90.000 deg
};
P[1729]{
   GP1:
	UF : 0, UT : 6,		CONFIG : 'N U T, 0, 0, 0',
	X =  58.976  mm,	Y =   -348.260  mm,	Z =   -252.761  mm,
	W =  90.000 deg,	P =   0.000 deg,	R =   90.000 deg
};
P[1730]{
   GP1:
	UF : 0, UT : 6,		CONFIG : 'N U T, 0, 0, 0',
	X =  59.921  mm,	Y =   -349.949  mm,	Z =   -252.578  mm,
	W =  90.000 deg,	P =   0.000 deg,	R =   90.000 deg
};
P[1731]{
   GP1:
	UF : 0, UT : 6,		CONFIG : 'N U T, 0, 0, 0',
	X =  60.899  mm,	Y =   -351.657  mm,	Z =   -252.520  mm,
	W =  90.000 deg,	P =   0.000 deg,	R =   90.000 deg
};
P[1732]{
   GP1:
	UF : 0, UT : 6,		CONFIG : 'N U T, 0, 0, 0',
	X =  61.640  mm,	Y =   -352.911  mm,	Z =   -252.629  mm,
	W =  90.000 deg,	P =   0.000 deg,	R =   90.000 deg
};
P[1733]{
   GP1:
	UF : 0, UT : 6,		CONFIG : 'N U T, 0, 0, 0',
	X =  63.521  mm,	Y =   -356.115  mm,	Z =   -252.820  mm,
	W =  90.000 deg,	P =   0.000 deg,	R =   90.000 deg
};
P[1734]{
   GP1:
	UF : 0, UT : 6,		CONFIG : 'N U T, 0, 0, 0',
	X =  64.432  mm,	Y =   -357.721  mm,	Z =   -252.719  mm,
	W =  90.000 deg,	P =   0.000 deg,	R =   90.000 deg
};
P[1735]{
   GP1:
	UF : 0, UT : 6,		CONFIG : 'N U T, 0, 0, 0',
	X =  64.903  mm,	Y =   -358.512  mm,	Z =   -252.813  mm,
	W =  90.000 deg,	P =   0.000 deg,	R =   90.000 deg
};
P[1736]{
   GP1:
	UF : 0, UT : 6,		CONFIG : 'N U T, 0, 0, 0',
	X =  65.410  mm,	Y =   -359.464  mm,	Z =   -252.545  mm,
	W =  90.000 deg,	P =   0.000 deg,	R =   90.000 deg
};
P[1737]{
   GP1:
	UF : 0, UT : 6,		CONFIG : 'N U T, 0, 0, 0',
	X =  67.161  mm,	Y =   -362.465  mm,	Z =   -252.661  mm,
	W =  90.000 deg,	P =   0.000 deg,	R =   90.000 deg
};
P[1738]{
   GP1:
	UF : 0, UT : 6,		CONFIG : 'N U T, 0, 0, 0',
	X =  67.625  mm,	Y =   -363.334  mm,	Z =   -252.424  mm,
	W =  90.000 deg,	P =   0.000 deg,	R =   90.000 deg
};
P[1739]{
   GP1:
	UF : 0, UT : 6,		CONFIG : 'N U T, 0, 0, 0',
	X =  68.421  mm,	Y =   -364.631  mm,	Z =   -252.719  mm,
	W =  90.000 deg,	P =   0.000 deg,	R =   90.000 deg
};
P[1740]{
   GP1:
	UF : 0, UT : 6,		CONFIG : 'N U T, 0, 0, 0',
	X =  69.158  mm,	Y =   -365.945  mm,	Z =   -252.584  mm,
	W =  90.000 deg,	P =   0.000 deg,	R =   90.000 deg
};
P[1741]{
   GP1:
	UF : 0, UT : 6,		CONFIG : 'N U T, 0, 0, 0',
	X =  70.581  mm,	Y =   -368.365  mm,	Z =   -252.737  mm,
	W =  90.000 deg,	P =   0.000 deg,	R =   90.000 deg
};
P[1742]{
   GP1:
	UF : 0, UT : 6,		CONFIG : 'N U T, 0, 0, 0',
	X =  72.170  mm,	Y =   -371.111  mm,	Z =   -252.763  mm,
	W =  90.000 deg,	P =   0.000 deg,	R =   90.000 deg
};
P[1743]{
   GP1:
	UF : 0, UT : 6,		CONFIG : 'N U T, 0, 0, 0',
	X =  73.583  mm,	Y =   -373.565  mm,	Z =   -252.741  mm,
	W =  90.000 deg,	P =   0.000 deg,	R =   90.000 deg
};
P[1744]{
   GP1:
	UF : 0, UT : 6,		CONFIG : 'N U T, 0, 0, 0',
	X =  74.077  mm,	Y =   -374.462  mm,	Z =   -252.586  mm,
	W =  90.000 deg,	P =   0.000 deg,	R =   90.000 deg
};
P[1745]{
   GP1:
	UF : 0, UT : 6,		CONFIG : 'N U T, 0, 0, 0',
	X =  74.514  mm,	Y =   -375.239  mm,	Z =   -252.519  mm,
	W =  90.000 deg,	P =   0.000 deg,	R =   90.000 deg
};
P[1746]{
   GP1:
	UF : 0, UT : 6,		CONFIG : 'N U T, 0, 0, 0',
	X =  76.059  mm,	Y =   -377.830  mm,	Z =   -252.824  mm,
	W =  90.000 deg,	P =   0.000 deg,	R =   90.000 deg
};
P[1747]{
   GP1:
	UF : 0, UT : 6,		CONFIG : 'N U T, 0, 0, 0',
	X =  77.200  mm,	Y =   -379.852  mm,	Z =   -252.656  mm,
	W =  90.000 deg,	P =   0.000 deg,	R =   90.000 deg
};
P[1748]{
   GP1:
	UF : 0, UT : 6,		CONFIG : 'N U T, 0, 0, 0',
	X =  79.231  mm,	Y =   -383.394  mm,	Z =   -252.565  mm,
	W =  90.000 deg,	P =   0.000 deg,	R =   90.000 deg
};
P[1749]{
   GP1:
	UF : 0, UT : 6,		CONFIG : 'N U T, 0, 0, 0',
	X =  79.674  mm,	Y =   -384.115  mm,	Z =   -252.735  mm,
	W =  90.000 deg,	P =   0.000 deg,	R =   90.000 deg
};
P[1750]{
   GP1:
	UF : 0, UT : 6,		CONFIG : 'N U T, 0, 0, 0',
	X =  81.294  mm,	Y =   -386.925  mm,	Z =   -252.722  mm,
	W =  90.000 deg,	P =   0.000 deg,	R =   90.000 deg
};
P[1751]{
   GP1:
	UF : 0, UT : 6,		CONFIG : 'N U T, 0, 0, 0',
	X =  81.596  mm,	Y =   -387.517  mm,	Z =   -252.479  mm,
	W =  90.000 deg,	P =   0.000 deg,	R =   90.000 deg
};
P[1752]{
   GP1:
	UF : 0, UT : 6,		CONFIG : 'N U T, 0, 0, 0',
	X =  82.587  mm,	Y =   -389.209  mm,	Z =   -252.561  mm,
	W =  90.000 deg,	P =   0.000 deg,	R =   90.000 deg
};
P[1753]{
   GP1:
	UF : 0, UT : 6,		CONFIG : 'N U T, 0, 0, 0',
	X =  83.684  mm,	Y =   -391.052  mm,	Z =   -252.766  mm,
	W =  90.000 deg,	P =   0.000 deg,	R =   90.000 deg
};
P[1754]{
   GP1:
	UF : 0, UT : 6,		CONFIG : 'N U T, 0, 0, 0',
	X =  84.262  mm,	Y =   -392.106  mm,	Z =   -252.576  mm,
	W =  90.000 deg,	P =   0.000 deg,	R =   90.000 deg
};
P[1755]{
   GP1:
	UF : 0, UT : 6,		CONFIG : 'N U T, 0, 0, 0',
	X =  84.830  mm,	Y =   -393.046  mm,	Z =   -252.733  mm,
	W =  90.000 deg,	P =   0.000 deg,	R =   90.000 deg
};
P[1756]{
   GP1:
	UF : 0, UT : 6,		CONFIG : 'N U T, 0, 0, 0',
	X =  85.269  mm,	Y =   -393.835  mm,	Z =   -252.627  mm,
	W =  90.000 deg,	P =   0.000 deg,	R =   90.000 deg
};
P[1757]{
   GP1:
	UF : 0, UT : 6,		CONFIG : 'N U T, 0, 0, 0',
	X =  85.641  mm,	Y =   -394.503  mm,	Z =   -252.540  mm,
	W =  90.000 deg,	P =   0.000 deg,	R =   90.000 deg
};
P[1758]{
   GP1:
	UF : 0, UT : 6,		CONFIG : 'N U T, 0, 0, 0',
	X =  86.256  mm,	Y =   -395.490  mm,	Z =   -252.822  mm,
	W =  90.000 deg,	P =   0.000 deg,	R =   90.000 deg
};
P[1759]{
   GP1:
	UF : 0, UT : 6,		CONFIG : 'N U T, 0, 0, 0',
	X =  87.337  mm,	Y =   -397.387  mm,	Z =   -252.732  mm,
	W =  90.000 deg,	P =   0.000 deg,	R =   90.000 deg
};
P[1760]{
   GP1:
	UF : 0, UT : 6,		CONFIG : 'N U T, 0, 0, 0',
	X =  88.973  mm,	Y =   -400.287  mm,	Z =   -252.500  mm,
	W =  90.000 deg,	P =   0.000 deg,	R =   90.000 deg
};
P[1761]{
   GP1:
	UF : 0, UT : 6,		CONFIG : 'N U T, 0, 0, 0',
	X =  89.381  mm,	Y =   -400.995  mm,	Z =   -252.498  mm,
	W =  90.000 deg,	P =   0.000 deg,	R =   90.000 deg
};
P[1762]{
   GP1:
	UF : 0, UT : 6,		CONFIG : 'N U T, 0, 0, 0',
	X =  89.757  mm,	Y =   -401.616  mm,	Z =   -252.599  mm,
	W =  90.000 deg,	P =   0.000 deg,	R =   90.000 deg
};
P[1763]{
   GP1:
	UF : 0, UT : 6,		CONFIG : 'N U T, 0, 0, 0',
	X =  90.672  mm,	Y =   -403.190  mm,	Z =   -252.638  mm,
	W =  90.000 deg,	P =   0.000 deg,	R =   90.000 deg
};
P[1764]{
   GP1:
	UF : 0, UT : 6,		CONFIG : 'N U T, 0, 0, 0',
	X =  91.252  mm,	Y =   -404.141  mm,	Z =   -252.833  mm,
	W =  90.000 deg,	P =   0.000 deg,	R =   90.000 deg
};
P[1765]{
   GP1:
	UF : 0, UT : 6,		CONFIG : 'N U T, 0, 0, 0',
	X =  94.477  mm,	Y =   -409.745  mm,	Z =   -252.766  mm,
	W =  90.000 deg,	P =   0.000 deg,	R =   90.000 deg
};
P[1766]{
   GP1:
	UF : 0, UT : 6,		CONFIG : 'N U T, 0, 0, 0',
	X =  94.906  mm,	Y =   -410.485  mm,	Z =   -252.769  mm,
	W =  90.000 deg,	P =   0.000 deg,	R =   90.000 deg
};
P[1767]{
   GP1:
	UF : 0, UT : 6,		CONFIG : 'N U T, 0, 0, 0',
	X =  95.504  mm,	Y =   -411.513  mm,	Z =   -252.796  mm,
	W =  90.000 deg,	P =   0.000 deg,	R =   90.000 deg
};
P[1768]{
   GP1:
	UF : 0, UT : 6,		CONFIG : 'N U T, 0, 0, 0',
	X =  97.112  mm,	Y =   -414.304  mm,	Z =   -252.778  mm,
	W =  90.000 deg,	P =   0.000 deg,	R =   90.000 deg
};
P[1769]{
   GP1:
	UF : 0, UT : 6,		CONFIG : 'N U T, 0, 0, 0',
	X =  98.564  mm,	Y =   -416.862  mm,	Z =   -252.630  mm,
	W =  90.000 deg,	P =   0.000 deg,	R =   90.000 deg
};
P[1770]{
   GP1:
	UF : 0, UT : 6,		CONFIG : 'N U T, 0, 0, 0',
	X =  99.540  mm,	Y =   -418.520  mm,	Z =   -252.739  mm,
	W =  90.000 deg,	P =   0.000 deg,	R =   90.000 deg
};
P[1771]{
   GP1:
	UF : 0, UT : 6,		CONFIG : 'N U T, 0, 0, 0',
	X =  100.891  mm,	Y =   -420.841  mm,	Z =   -252.803  mm,
	W =  90.000 deg,	P =   0.000 deg,	R =   90.000 deg
};
P[1772]{
   GP1:
	UF : 0, UT : 6,		CONFIG : 'N U T, 0, 0, 0',
	X =  101.236  mm,	Y =   -421.448  mm,	Z =   -252.772  mm,
	W =  90.000 deg,	P =   0.000 deg,	R =   90.000 deg
};
P[1773]{
   GP1:
	UF : 0, UT : 6,		CONFIG : 'N U T, 0, 0, 0',
	X =  101.650  mm,	Y =   -422.257  mm,	Z =   -252.442  mm,
	W =  90.000 deg,	P =   0.000 deg,	R =   90.000 deg
};
P[1774]{
   GP1:
	UF : 0, UT : 6,		CONFIG : 'N U T, 0, 0, 0',
	X =  103.191  mm,	Y =   -424.911  mm,	Z =   -252.501  mm,
	W =  90.000 deg,	P =   0.000 deg,	R =   90.000 deg
};
P[1775]{
   GP1:
	UF : 0, UT : 6,		CONFIG : 'N U T, 0, 0, 0',
	X =  103.560  mm,	Y =   -425.577  mm,	Z =   -252.403  mm,
	W =  90.000 deg,	P =   0.000 deg,	R =   90.000 deg
};
P[1776]{
   GP1:
	UF : 0, UT : 6,		CONFIG : 'N U T, 0, 0, 0',
	X =  104.143  mm,	Y =   -426.540  mm,	Z =   -252.572  mm,
	W =  90.000 deg,	P =   0.000 deg,	R =   90.000 deg
};
P[1777]{
   GP1:
	UF : 0, UT : 6,		CONFIG : 'N U T, 0, 0, 0',
	X =  104.631  mm,	Y =   -427.327  mm,	Z =   -252.778  mm,
	W =  90.000 deg,	P =   0.000 deg,	R =   90.000 deg
};
P[1778]{
   GP1:
	UF : 0, UT : 6,		CONFIG : 'N U T, 0, 0, 0',
	X =  104.983  mm,	Y =   -428.000  mm,	Z =   -252.549  mm,
	W =  90.000 deg,	P =   0.000 deg,	R =   90.000 deg
};
P[1779]{
   GP1:
	UF : 0, UT : 6,		CONFIG : 'N U T, 0, 0, 0',
	X =  105.394  mm,	Y =   -428.731  mm,	Z =   -252.483  mm,
	W =  90.000 deg,	P =   0.000 deg,	R =   90.000 deg
};
P[1780]{
   GP1:
	UF : 0, UT : 6,		CONFIG : 'N U T, 0, 0, 0',
	X =  106.902  mm,	Y =   -431.311  mm,	Z =   -252.595  mm,
	W =  90.000 deg,	P =   0.000 deg,	R =   90.000 deg
};
P[1781]{
   GP1:
	UF : 0, UT : 6,		CONFIG : 'N U T, 0, 0, 0',
	X =  109.075  mm,	Y =   -435.104  mm,	Z =   -252.490  mm,
	W =  90.000 deg,	P =   0.000 deg,	R =   90.000 deg
};
P[1782]{
   GP1:
	UF : 0, UT : 6,		CONFIG : 'N U T, 0, 0, 0',
	X =  109.728  mm,	Y =   -436.176  mm,	Z =   -252.698  mm,
	W =  90.000 deg,	P =   0.000 deg,	R =   90.000 deg
};
P[1783]{
   GP1:
	UF : 0, UT : 6,		CONFIG : 'N U T, 0, 0, 0',
	X =  110.181  mm,	Y =   -436.936  mm,	Z =   -252.782  mm,
	W =  90.000 deg,	P =   0.000 deg,	R =   90.000 deg
};
P[1784]{
   GP1:
	UF : 0, UT : 6,		CONFIG : 'N U T, 0, 0, 0',
	X =  110.980  mm,	Y =   -438.336  mm,	Z =   -252.730  mm,
	W =  90.000 deg,	P =   0.000 deg,	R =   90.000 deg
};
P[1785]{
   GP1:
	UF : 0, UT : 6,		CONFIG : 'N U T, 0, 0, 0',
	X =  111.527  mm,	Y =   -439.315  mm,	Z =   -252.622  mm,
	W =  90.000 deg,	P =   0.000 deg,	R =   90.000 deg
};
P[1786]{
   GP1:
	UF : 0, UT : 6,		CONFIG : 'N U T, 0, 0, 0',
	X =  112.100  mm,	Y =   -440.264  mm,	Z =   -252.777  mm,
	W =  90.000 deg,	P =   0.000 deg,	R =   90.000 deg
};
P[1787]{
   GP1:
	UF : 0, UT : 6,		CONFIG : 'N U T, 0, 0, 0',
	X =  112.499  mm,	Y =   -441.063  mm,	Z =   -252.382  mm,
	W =  90.000 deg,	P =   0.000 deg,	R =   90.000 deg
};
P[1788]{
   GP1:
	UF : 0, UT : 6,		CONFIG : 'N U T, 0, 0, 0',
	X =  113.396  mm,	Y =   -442.537  mm,	Z =   -252.670  mm,
	W =  90.000 deg,	P =   0.000 deg,	R =   90.000 deg
};
P[1789]{
   GP1:
	UF : 0, UT : 6,		CONFIG : 'N U T, 0, 0, 0',
	X =  113.755  mm,	Y =   -443.192  mm,	Z =   -252.555  mm,
	W =  90.000 deg,	P =   0.000 deg,	R =   90.000 deg
};
P[1790]{
   GP1:
	UF : 0, UT : 6,		CONFIG : 'N U T, 0, 0, 0',
	X =  116.745  mm,	Y =   -448.315  mm,	Z =   -252.750  mm,
	W =  90.000 deg,	P =   0.000 deg,	R =   90.000 deg
};
P[1791]{
   GP1:
	UF : 0, UT : 6,		CONFIG : 'N U T, 0, 0, 0',
	X =  118.445  mm,	Y =   -451.289  mm,	Z =   -252.650  mm,
	W =  90.000 deg,	P =   0.000 deg,	R =   90.000 deg
};
P[1792]{
   GP1:
	UF : 0, UT : 6,		CONFIG : 'N U T, 0, 0, 0',
	X =  120.375  mm,	Y =   -454.613  mm,	Z =   -252.708  mm,
